// ---- POUs/Machine/UV_LED_Modul/FB_UvLedModule.TcPOU
FUNCTION_BLOCK FB_UvLedModule IMPLEMENTS I_DeviceBase
VAR_INPUT
  IbReady                  AT%I* : BOOL;
END_VAR

VAR_OUTPUT
  ObEnableHigh             AT%Q* : BOOL;
  ObLowIntenseMode         AT%Q* : BOOL;
  ObDisableLeft            AT%Q* : BOOL;
  ObDisableRight           AT%Q* : BOOL;
  OnIntensitySetpoint      AT%Q* : WORD;  (*Setpoint for intensity control  [digit]*)
END_VAR

VAR
  _bActivate                     : BOOL;
  _sName                         : STRING := '';
  _nColorRGB                     : UDINT;
  _sColorName                    : STRING := 'undef';    (*color name*)
END_VAR

VAR CONSTANT
  CnAnalogMinDigit               : DINT := 0;      (*Min value analog-output in digit*)
  CnAnalogMaxDigit               : DINT := 32767;  (*Max value analog-output in digit*)
  CnMinIntensitySetpoint         : DINT := 5;      (*Min setpoint for intensity control [%]*)
  CnMaxIntensitySetpoint         : DINT := 100;    (*Max setpoint for intensity control [%]*)
END_VAR

VAR PERSISTENT
  RbLowIntenseMode               : BOOL := FALSE;  (*Visu: set low intense mode*)
  RbDisableLeft                  : BOOL := FALSE;  (*Visu: disable left SLM*)
  RbDisableRight                 : BOOL := FALSE;  (*Visu: disable right SLM*)
  RnIntensitySetpoint            : DINT := 20;     (*Visu: setpoint for intensity control [%]*)
END_VAR

(*Set outputs*)
ObEnableHigh        := _bActivate;
ObLowIntenseMode    := RbLowIntenseMode;
ObDisableLeft       := RbDisableLeft;
ObDisableRight      := RbDisableRight;
OnIntensitySetpoint := DINT_TO_WORD(CnAnalogMaxDigit * RnIntensitySetpoint / 100);  (*Setpoint [digit]*)

METHOD Init : BOOL
VAR_INPUT
  nColorRGB    : UDINT;     (*color RGB*)
  sColorName   : STRING;    (*color name*)
END_VAR
_nColorRGB := nColorRGB;
_sColorName := sColorName;
END_METHOD

METHOD mDisable : BOOL
_bActivate := FALSE;
END_METHOD

METHOD mEnable : BOOL
_bActivate := TRUE;
END_METHOD

{attribute 'monitoring':='call'}
PROPERTY pActive : BOOL
GET
pActive := _bActivate;
END_GET
END_PROPERTY

PROPERTY pErrorCode : INT
GET
pErrorCode := 0;  // no error
END_GET
END_PROPERTY

END_FUNCTION_BLOCK

// ---- POUs/Print/Ads/FB_ADS_CAMERA.TcPOU
FUNCTION_BLOCK FB_ADS_CAMERA EXTENDS FB_AdsBlockBase
VAR
  stAds : ST_ADS_CAMERA;
END_VAR



// Todo redirect PucPath to internal sAdsStruct instead of fb Instance
// - write InstanceName
// - or override getPucPath() (but is PRIVATE)

// The output variables are not used, please add eaccessors if needed
(*
 (*Out*)
  iO_MaxNbMarksQV           : INT := GVL_Camera.cC_QUALIVISION_MAX_NB_MARKS; 
  sO_PointsReadQV           : ST_COMMAND_PLC;    (*New points read by QualiVision*)
  iO_AvailableNbReadPointQV : INT; 
  sO_ReadPointsQV           : ARRAY[1..GVL_Camera.cC_QUALIVISION_MAX_NB_MARKS] OF ST_CAMERA_CORRECTION_QV;
*)

{attribute 'monitoring' := 'call'}
(*
  Name of the block. 
  A friendly name (which is used in the PUC to show the element (only for some blocks/apps))
*)
PROPERTY aName : T_MaxString
GET
aName := aO_Name;
END_GET
SET
aO_Name := aName;
stAds.aO_Name := aName; // update in struct as well
END_SET
END_PROPERTY

PROPERTY bEnable : BOOL
GET
bEnable   := stAds.bI_Enable;   // Set ads interface variable
END_GET
SET
stAds.bI_Enable := bEnable;   // set interface variable
END_SET
END_PROPERTY

METHOD config
VAR_INPUT

END_VAR

//initRemVar();
END_METHOD

PROPERTY eCameraDevice : E_CameraDevice
GET
eCameraDevice := stAds.eI_CameraDevice;
END_GET
SET
stAds.eI_CameraDevice := eCameraDevice;
END_SET
END_PROPERTY

PROPERTY eCameraMode : E_CameraMode
GET
eCameraMode := stAds.eI_CameraMode;
END_GET
SET
stAds.eI_CameraMode := eCameraMode;
END_SET
END_PROPERTY

PROPERTY eTeachProgress : EN_CAMERA_TEACH
GET
eTeachProgress := stAds.eI_TeachProgress;
END_GET
END_PROPERTY

METHOD PROTECTED getPucPath : STRING
VAR
END_VAR
// apply puc path to struct (instead of fb declaraion)
getPucPath := F_Concat3(SUPER^.getPucPath(), '.', 'stAds');
END_METHOD

PROPERTY pCorrectionPointsIndication : POINTER TO ARRAY[1..4] OF ST_CORRECTION_POINT;
GET
pCorrectionPointsIndication := ADR(stAds.sI_CorrectionPointIndication);
END_GET
END_PROPERTY

PROPERTY pTeachPointsQV : POINTER TO ARRAY[1..GVL_Camera.cC_QUALIVISION_MAX_NB_MARKS] OF ST_CAMERA_TEACH_QV;
GET
pTeachPointsQV := ADR(stAds.sI_TeachPointsQV);
END_GET
END_PROPERTY

(*
  Setup constant ADS Block definitions.
  HOWTO: in abstract implmentation call
      init(aVersion:=, aType:=, nType:=, eLayer:=);
*)
METHOD  setup

init(aVersion:=convertVersionIntToString(stAds.iO_Version), aType:=stAds.aO_Type, nType:=ePr_BLK_CAMERA, eLayer:=E_AdsLayer.Structural);
END_METHOD

PROPERTY sMsgInterface : POINTER TO ST_ADS_MSG_IF
GET
sMsgInterface := ADR(stAds.sO_Message);
END_GET
END_PROPERTY

END_FUNCTION_BLOCK

// ---- POUs/Print/Ads/FB_ADS_DVTSHEETALIGNMENT.TcPOU
FUNCTION_BLOCK FB_ADS_DVTSHEETALIGNMENT EXTENDS FB_AdsBlockBase
VAR
  // ---------------------------------
  // ADS interface block specific
  sO_Message         : ST_ADS_MSG_IF;
  
  bI_Enable          : BOOL := TRUE;    (*Enable processing*)

  bI_UsePrintMark    : BOOL := TRUE;    (*Enable processing of print marks*)
  sI_PrintMarkSizeX  : ST_VAR_IN_REAL;  (*Print mark X size [mm]*)
  sI_PrintMarkSizeY  : ST_VAR_IN_REAL;  (*Print mark Y size [mm]*)

  sI_HeadGap         : ST_VAR_IN_REAL;  (*Gap between head and substrate [mm]*)

  lI_SegmentSize     : UDINT;           (*Distance between two images in pixel*)
  lI_SegmentCount    : UDINT;           (*Number of images*)
  fI_SegmentAngle    : REAL;            (*Angle between two segments in deg*)

  sI_DeltaX          : ST_VAR_IN_REAL;  (*X offset between camera marks [mm]*)

  bI_IsMaintenanceJob: BOOL;            (*Maintenance job: disable shift and rotation*)

  (*Out*)
  sO_CurrentAngle    : ST_VAR_OUT_REAL; (*Last measured angle in deg*)
  lO_CurrentYShift   : UDINT;           (*Last measured Y Shift in Pixel*)

  bO_RangeErrorAngle : BOOL;            (*Measured angle out of range*)
  bO_RangeErrorShift : BOOL;            (*Measured shift out of range*)

  // ---------------------------------
END_VAR
VAR PERSISTENT
  aR_Pattern         : UDINT;           (*check pattern for rem validity*)
  bR_Enable          : BOOL;            (*remanent: *)
  bR_UsePrintMark    : BOOL;            (*remanent: *)
  fR_PrintMarkSize_X : REAL;            (*remanent: *)
  fR_PrintMarkSize_Y : REAL;            (*remanent: *)
  fR_HeadGap         : REAL;            (*remanent: head gap in [mm]*)
  fR_DeltaX          : REAL;            (*remanent: *)
END_VAR

PROPERTY bEnable : BOOL
GET
bEnable   := bI_Enable;   // Set ads interface variable
bR_Enable := bI_Enable;   // Update remanent variable
END_GET
SET
bI_Enable := bEnable;   // set interface variable
bR_Enable := bEnable;   // update remanent variable
END_SET
END_PROPERTY

PROPERTY bIsMaintenanceJob : BOOL
GET
bIsMaintenanceJob := bI_IsMaintenanceJob;   // Set ads interface variable
END_GET
SET
bI_IsMaintenanceJob := bIsMaintenanceJob;   // Set ads interface variable
END_SET
END_PROPERTY

PROPERTY bRangeErrorAngle : BOOL
SET
bO_RangeErrorAngle := bRangeErrorAngle;
END_SET
END_PROPERTY

PROPERTY bRangeErrorShift : BOOL
SET
bO_RangeErrorShift := bRangeErrorShift;
END_SET
END_PROPERTY

PROPERTY bUsePrintMark : BOOL
GET
bUsePrintMark   := bI_UsePrintMark;   // Set ads interface variable
bR_UsePrintMark := bI_UsePrintMark;   // Update remanent variable
END_GET
SET
bI_UsePrintMark := bUsePrintMark;   // set interface variable
bR_UsePrintMark := bUsePrintMark;   // update remanent variable
END_SET
END_PROPERTY

METHOD config
VAR_INPUT
  bPrintMarkSizeX_Exist : BOOL;
  aPrintMarkSizeX_Unit  : STRING;
  fPrintMarkSizeX_Min   : REAL;
  fPrintMarkSizeX_Max   : REAL;
  
  bPrintMarkSizeY_Exist : BOOL;
  aPrintMarkSizeY_Unit  : STRING;
  fPrintMarkSizeY_Min   : REAL;
  fPrintMarkSizeY_Max   : REAL;
  
  bHeadGap_Exist        : BOOL;
  aHeadGap_Unit         : STRING;
  fHeadGap_Min          : REAL;
  fHeadGap_Max          : REAL;

  bDeltaX_Exist         : BOOL;
  aDeltaX_Unit          : STRING;
  fDeltaX_Min           : REAL;
  fDeltaX_Max           : REAL;
  
  bCurrentAngle_Exist   : BOOL;
  aCurrentAngle_Unit    : STRING;
  fCurrentAngle_Min     : REAL;
  fCurrentAngle_Max     : REAL;
END_VAR
sI_PrintMarkSizeX.bC_Exist := bPrintMarkSizeX_Exist;
sI_PrintMarkSizeX.aC_Unit  := aPrintMarkSizeX_Unit;
sI_PrintMarkSizeX.fC_Min   := fPrintMarkSizeX_Min;
sI_PrintMarkSizeX.fC_Max   := fPrintMarkSizeX_Max;
sI_PrintMarkSizeY.bC_Exist := bPrintMarkSizeY_Exist;
sI_PrintMarkSizeY.aC_Unit  := aPrintMarkSizeY_Unit;
sI_PrintMarkSizeY.fC_Min   := fPrintMarkSizeY_Min;
sI_PrintMarkSizeY.fC_Max   := fPrintMarkSizeY_Max;
sI_HeadGap.bC_Exist        := bHeadGap_Exist;
sI_HeadGap.aC_Unit         := aHeadGap_Unit;
sI_HeadGap.fC_Min          := fHeadGap_Min;
sI_HeadGap.fC_Max          := fHeadGap_Max;
sI_DeltaX.bC_Exist         := bDeltaX_Exist;
sI_DeltaX.aC_Unit          := aDeltaX_Unit;
sI_DeltaX.fC_Min           := fDeltaX_Min;
sI_DeltaX.fC_Max           := fDeltaX_Max;
sO_CurrentAngle.bC_Exist   := bCurrentAngle_Exist;
sO_CurrentAngle.aC_Unit    := aCurrentAngle_Unit;
sO_CurrentAngle.fC_Min     := fCurrentAngle_Min;
sO_CurrentAngle.fC_Max     := fCurrentAngle_Max;

sO_CurrentAngle.bC_Exist   := FALSE;

initRemVar();
END_METHOD

PROPERTY fDeltaX : REAL
GET
fDeltaX   := sI_DeltaX.fI_Val;   // Set ads interface variable
fR_DeltaX := sI_DeltaX.fI_Val;
END_GET
END_PROPERTY

// HeadGap in [mm]
PROPERTY fHeadGap : LREAL
GET
fHeadGap   := sI_HeadGap.fI_Val;   // Set ads interface variable
fR_HeadGap := sI_HeadGap.fI_Val;   // Update remanent variable
END_GET
SET
sI_HeadGap.fI_Val := TO_REAL(fHeadGap);   // set interface variable
fR_HeadGap        := TO_REAL(fHeadGap);   // update remanent variable
END_SET
END_PROPERTY

PROPERTY fMarkSizeX : REAL
GET
fMarkSizeX         := sI_PrintMarkSizeX.fI_Val;   // Set ads interface variable
fR_PrintMarkSize_X := sI_PrintMarkSizeX.fI_Val;   // Update remanent variable
END_GET
END_PROPERTY

PROPERTY fMarkSizeY : REAL
GET
fMarkSizeY         := sI_PrintMarkSizeY.fI_Val;   // Set ads interface variable
fR_PrintMarkSize_Y := sI_PrintMarkSizeY.fI_Val;   // Update remanent variable
END_GET
END_PROPERTY

PROPERTY fO_CurrentAngle : LREAL
SET
sO_CurrentAngle.fO_Val := tO_REAL(fO_CurrentAngle);
END_SET
END_PROPERTY

PROPERTY fSegmentAngle : REAL
GET
fSegmentAngle := fI_SegmentAngle;   // Set ads interface variable
END_GET
END_PROPERTY

METHOD PROTECTED initRemVar
(*load default initial values if pattern was invalid*)
IF aR_Pattern <> 16#ABCD THEN
  aR_Pattern  := 16#ABCD;  
  bR_Enable   := TRUE;
  bR_UsePrintMark := 0;
  fR_PrintMarkSize_X := 0;
  fR_PrintMarkSize_Y := 0;
  fR_HeadGap  := 2;
  fR_DeltaX := 0;
END_IF

bI_Enable := bR_Enable;
bI_UsePrintMark := bR_UsePrintMark;
sI_PrintMarkSizeX.fI_Val := fR_PrintMarkSize_X;
sI_PrintMarkSizeY.fI_Val := fR_PrintMarkSize_Y;
sI_HeadGap.fI_Val := fR_HeadGap;
sI_DeltaX.fI_Val := fR_DeltaX;
END_METHOD

PROPERTY nO_CurrentYShift : UDINT
SET
lO_CurrentYShift := nO_CurrentYShift;
END_SET
END_PROPERTY

PROPERTY nSegmentCount : UDINT
GET
nSegmentCount := lI_SegmentCount;   // Set ads interface variable
END_GET
END_PROPERTY

PROPERTY nSegmentSize : UDINT
GET
nSegmentSize := lI_SegmentSize;   // Set ads interface variable
END_GET
END_PROPERTY

(*
  Setup constant ADS Block definitions.
  HOWTO: in abstract implmentation call
      init(aVersion:=, aType:=, nType:=, eLayer:=);
*)
METHOD  setup
init(aVersion:='01.00.10', aType:='DvtSheetAlignment', nType:=ePr_BLK_SA, eLayer:=E_AdsLayer.Structural);
END_METHOD

PROPERTY sMsgInterface : POINTER TO ST_ADS_MSG_IF
GET
sMsgInterface := ADR(sO_Message);
END_GET
END_PROPERTY

END_FUNCTION_BLOCK

// ---- POUs/Print/Camera/FB_CameraBase.TcPOU
(*
  Base camera system
  Implements I_Camera: set I_CameraSink.   
*)
FUNCTION_BLOCK ABSTRACT FB_CameraBase EXTENDS FB_Commons IMPLEMENTS I_Camera, I_CameraTriggerDevice

VAR
  _bInitialized             : BOOL;
  _iCameraSink              : I_CameraSink;
  _iCameraTrigger           : I_CameraTrigger;
  _bSimulate                : BOOL;
  _nPrintUnitResolution     : UDINT;           (*printhead pixel resolution [dpi]*)
  _nPrintUnitSubPx          : UDINT;           (*print unit SubPixel resolution [SubPx]*)
  _bUseCameraTrigger        : BOOL;            (*use a trigger output timestamp I/O*)
  _bUseCameraTriggerFeedback : BOOL;           (*use a camera triggered feedback timestamp I/O*)
  _eCameraMode              : E_CameraMode;    (*desired camera mode*)
  _ePossibleMode            : E_CameraMode;    (*currently possible mode*)
  _fSubstrateLength         : LREAL := 1;      (*Substrate length [m]*)
  _fSubstrateWidth          : LREAL := 1;      (*Substrate width [m]*)
  _fImageLength             : LREAL := 1;      (*Image length [m]*)
  _fImageWidth              : LREAL := 1;      (*Image width [m]*)
  _fFrameLength             : LREAL := 1;      (*Camera Frame width in [px]*)
  _bActivated               : BOOL;            (*Camera is activated*)
  _sVisuName                : STRING := 'unvailable';     (*detail visualisation instance name*)
  
  // status
  _bCamTriggerOk            : BOOL;
  _bCamTriggerStarted       : BOOL;
  _bCamTriggerDone          : BOOL;   
  _nCamStartPos             : DINT;            (*Cam start position ideal [SubPx]*)
  _nCamStartPosDeviation    : DINT;            (*Cam stated position real [SubPx]*)
  _nRxCamPoints             : UDINT;           (*number of received cam points*)

  // helper
  stCamPoint                : ST_DeformationPointAccurate;(*actual camera point*)
    
  // messaging
  _pMsgConfig               : POINTER TO CalmarCommons.ST_MSG_CONFIG;
END_VAR

VAR PERSISTENT
  _fTriggerDistance         : LREAL;           (*[m] Distance between Sensor and Trigger*)
  _fTriggerPulseLength      : LREAL := 10;     (*[ms] Length of trigger signal in ms, min. 3 bus cycles*)
  _fDetectToCameraOffset    : LREAL := 0.1;    (*[m] Distance between input trigger and camera, mech.*)
  _fCameraToPrintOffset     : LREAL := 0.0;    (*[m] Distance between Camera and PU, mech, This offset can be used to shift the reference of a camera/sheet-detect, e.g. because this reference is different from to one where the alignment Camera/sheetdetect-PrintUnit has been made*)
END_VAR

METHOD ActivateCam : BOOL
VAR_INPUT
  iCameraSink : I_CameraSink;
END_VAR
IF iCameraSink = 0 THEN
  LogError('Invalid parameter (0 pointer)');
  ActivateCam := FALSE;
  RETURN; 
ELSIF _iCameraSink <> 0 AND iCameraSink <>_iCameraSink THEN
  LogError('SetSink failed: other sink already exists');
  ActivateCam := FALSE;
  RETURN; 
END_IF 

_iCameraSink := iCameraSink;
_iCameraTrigger.Enable(iCam:=THIS^, bUseCameraTrigger:=_bUseCameraTrigger, bUseCameraTriggerFeedback:=_bUseCameraTriggerFeedback);

_bActivated := TRUE;
ActivateCam:=TRUE;
END_METHOD

(*
  Activate/Deactivate camera trigger device
*)
PROPERTY bEnableTrigger : BOOL
SET
IF bEnableTrigger THEN
  _iCameraTrigger.Enable(iCam := THIS^, bUseCameraTrigger:= _bUseCameraTrigger, bUseCameraTriggerFeedback:=_bUseCameraTriggerFeedback);
ELSE
  _iCameraTrigger.Disable();
END_IF
END_SET
END_PROPERTY

(*
  Activate/Deactivate camera manual teach mode
*)
PROPERTY bManualTeach : BOOL
SET
_iCameraTrigger.bManualTeach := bManualTeach;
END_SET
END_PROPERTY

{attribute 'monitoring':='call'}
PROPERTY bSimulate : BOOL
GET
bSimulate := _bSimulate;
END_GET
SET
_bSimulate := bSimulate;
END_SET
END_PROPERTY

METHOD CamTrigger
VAR_INPUT
  bOk             : BOOL;     // trigger is ok
	nPos            : DINT;     // camera triggered position
  nPosDeviation   : DINT;     // camera started deviation
  nX0             : DINT;     // detected position sheet/repetition
END_VAR
_nRxCamPoints := 0;
_bCamTriggerStarted    := TRUE;
_bCamTriggerDone       := FALSE;
_bCamTriggerOk  := bOk;
_nCamStartPos   := nPos;
_nCamStartPosDeviation := nPosDeviation;

LogLvl(Lvl:=E_LogSeverity.Debug, Msg:=F_Concat2('CamTrigger at X0=', TO_STRING(nPos)));
IF _iCameraSink <> 0 THEN   // inform sink
  _iCameraSink.CamStarted(nX0:=nX0);
END_IF
END_METHOD

METHOD CamTriggerDone
_bCamTriggerStarted    := FALSE;  // this call marks the end of the camera trigger period
_bCamTriggerDone       := TRUE;

LogLvl(Lvl:=E_LogSeverity.Debug, Msg:='CamTriggerDone');
IF _iCameraSink <> 0 THEN   // inform sink
  _iCameraSink.CamDone();
END_IF
END_METHOD

METHOD DeactivateCam : BOOL
VAR_INPUT
  iSink : I_CameraSink;
END_VAR
IF _iCameraSink <> 0 AND iSink <> _iCameraSink THEN
  LogError('remove sink failed: inconsistent');
  DeactivateCam := FALSE;
  RETURN;  
END_IF

_iCameraSink := 0;
_iCameraTrigger.Disable();
_bActivated := FALSE;
DeactivateCam:=TRUE;
END_METHOD

{attribute 'monitoring':='call'}
PROPERTY ABSTRACT eCameraMode : E_CameraMode
GET
END_GET
END_PROPERTY

{attribute 'monitoring':='call'}
PROPERTY ABSTRACT eDeviceType : E_CameraDevice
GET
END_GET
END_PROPERTY

{attribute 'monitoring':='call'}
PROPERTY fCameraToPrintOffset : LREAL
GET
//This offset can be used to shift the reference of a camera, e.g. because this reference is different from to one where the alignment Camera-PrintUnit has been made
fCameraToPrintOffset := _fCameraToPrintOffset;
END_GET
SET
_fCameraToPrintOffset := fCameraToPrintOffset;
END_SET
END_PROPERTY

{attribute 'monitoring':='call'}
PROPERTY fDetectToCameraOffset : LREAL
GET
//This offset can be used to shift the reference of a camera, e.g. because this reference is different from to one where the alignment Camera-PrintUnit has been made
fDetectToCameraOffset := _fDetectToCameraOffset;
END_GET
SET
_fDetectToCameraOffset := fDetectToCameraOffset;
END_SET
END_PROPERTY

{attribute 'monitoring':='call'}
(* camera frame size in [px]*)
PROPERTY fFrameLength : LREAL
GET
fFrameLength := _fFrameLength;
END_GET
SET
_fFrameLength := fFrameLength;
END_SET
END_PROPERTY

{attribute 'monitoring':='call'}
(*Image Length/Depth in [m]*)
PROPERTY fImageLength : LREAL
GET
fImageLength := _fImageLength;
END_GET
SET
_fImageLength := fImageLength;
END_SET
END_PROPERTY

{attribute 'monitoring':='call'}
(*Image Width in [m]*)
PROPERTY fImageWidth : LREAL
GET
fImageWidth := _fImageWidth;
END_GET
SET
_fImageWidth := fImageWidth;
END_SET
END_PROPERTY

{attribute 'monitoring':='call'}
(*Substrate Length/Depth in [m]*)
PROPERTY fSubstrateLength : LREAL
GET
fSubstrateLength := _fSubstrateLength;
END_GET
SET
//ROI in Print direction
IF _iCameraTrigger <> 0 THEN
  _iCameraTrigger.SetSubstrateLength(fSubstrateLength := fSubstrateLength);   // save to camera trigger
  _fSubstrateLength := fSubstrateLength;                                      // save to camera
END_IF
END_SET
END_PROPERTY

{attribute 'monitoring':='call'}
(*Substrate Width in [m]*)
PROPERTY fSubstrateWidth : LREAL
GET
fSubstrateWidth := _fSubstrateWidth;
END_GET
SET
_fSubstrateWidth := fSubstrateWidth;
END_SET
END_PROPERTY

{attribute 'monitoring':='call'}
PROPERTY fTriggerDistance : LREAL
GET
fTriggerDistance := _fTriggerDistance;
END_GET
SET
_fTriggerDistance := fTriggerDistance;
END_SET
END_PROPERTY

PROPERTY fTriggerPulseLength : LREAL
GET
fTriggerPulseLength := _fTriggerPulseLength;
END_GET
END_PROPERTY

METHOD ABSTRACT GetCamStatus : BOOL
VAR_OUTPUT
  bConnectionOK  : BOOL;    // Camera connected
  bTeachOk       : BOOL;    // Teach successful
  nTeachedPoints : UDINT;   // Teached points for this job
  nScannedPoints : UDINT;   // Scanned points on current sheet  
  bCamStarted    : BOOL;    // Camera trigger is active, cam started
  bCamDone       : BOOL;    // Camera finished on last CT
  bErrors        : ARRAY[1..GVL_Camera.nC_NbCamErrors] OF BOOL;  // generic error flag list
END_VAR
END_METHOD

METHOD Init
VAR_INPUT
  nPrintUnitResolution         : UDINT;    (*printhead pixel resolution [dpi]*)
  nPrintUnitSubPx              : UDINT;    (*print unit subPixel resolution [SubPx]*)
  iCameraTrigger               : I_CameraTrigger;
  bUseCameraTrigger            : BOOL;     (*use a trigger output timestamp I/O*)
  bUseCameraTriggerFeedback    : BOOL;     (*use a camera triggered feedback timestamp I/O*)
END_VAR
IF nPrintUnitResolution <> 0 AND iCameraTrigger <> 0 THEN
  _nPrintUnitResolution := nPrintUnitResolution;
  _nPrintUnitSubPx      := nPrintUnitSubPx;
  _iCameraTrigger       := iCameraTrigger;
  
  _bUseCameraTrigger := bUseCameraTrigger;
  _bUseCameraTriggerFeedback := bUseCameraTriggerFeedback;
  
  _bInitialized := TRUE;
ELSE
  _bInitialized := FALSE;
END_IF
END_METHOD

METHOD mJobStart : BOOL
END_METHOD

(*
  Set mode to camera.
  :return: TRUE if success
*)
METHOD ABSTRACT setCameraMode : BOOL
VAR_INPUT
  eCameraMode : E_CameraMode;
END_VAR
END_METHOD

METHOD setMsgInterface : BOOL
VAR_INPUT
	pMsgConfig	: POINTER TO CalmarCommons.ST_MSG_CONFIG;
END_VAR
_pMsgConfig := pMsgConfig;
END_METHOD

{attribute 'monitoring':='call'}
PROPERTY sName : STRING
GET
sName := 'undefined';
END_GET
END_PROPERTY

{attribute 'monitoring':='call'}
PROPERTY sVisuName : STRING
GET
sVisuName := _sVisuName;
END_GET
SET
_sVisuName := sVisuName;
END_SET
END_PROPERTY

END_FUNCTION_BLOCK

// ---- POUs/Print/Camera/FB_CameraDummy.TcPOU
FUNCTION_BLOCK FB_CameraDummy EXTENDS FB_CameraBase
VAR_INPUT
END_VAR
VAR_OUTPUT
END_VAR
VAR
END_VAR

{attribute 'monitoring':='call'}
PROPERTY eCameraMode : E_CameraMode
GET
eCameraMode := _eCameraMode;
IF _eCameraMode = E_CameraMode.Auto THEN
  eCameraMode := E_CameraMode.NoCorrection;
END_IF
END_GET
END_PROPERTY

PROPERTY eDeviceType : E_CameraDevice
GET
eDeviceType := E_CameraDevice.SheetDetect;
END_GET
END_PROPERTY

METHOD GetCamStatus : BOOL
VAR_OUTPUT
  bConnectionOK  : BOOL;    // Camera connected
  bTeachOk       : BOOL;    // Teach successful
  nTeachedPoints : UDINT;   // Teached points for this job
  nScannedPoints : UDINT;   // Scanned points on current sheet
  bCamStarted    : BOOL;    // Camera trigger is active, cam started
  bCamDone       : BOOL;    // Camera finished on last CT
  bErrors        : ARRAY[1..GVL_Camera.nC_NbCamErrors] OF BOOL;  // generic error flag list
END_VAR
bConnectionOK  := TRUE;  //NO comm with a cam 
bTeachOk       := TRUE;  //NO teach availabe
nTeachedPoints := 0;
nScannedPoints := 0;
bCamStarted    := _bCamTriggerStarted;
bCamDone       := _bCamTriggerDone;

GetCamStatus := TRUE;
END_METHOD

(*
  Set mode to camera.
  :return: TRUE if success
*)
METHOD setCameraMode : BOOL
VAR_INPUT
  eCameraMode : E_CameraMode;
END_VAR
IF eCameraMode = E_CameraMode.NoCorrection THEN   // supported mode
  
  _eCameraMode := eCameraMode; 
  setCameraMode := TRUE;        // set desired mode
ELSE
  LogError(F_Concat3('Camera mode=', TO_STRING(eCameraMode), ' not supported by camera'));
  _eCameraMode := E_CameraMode.NoCorrection;
END_IF
END_METHOD

{attribute 'monitoring':='variable'}
PROPERTY sName : STRING
GET
sName := 'SheetDetect';
END_GET
END_PROPERTY

END_FUNCTION_BLOCK

// ---- POUs/Print/Camera/FB_CameraTcpIp.TcPOU
(*
  Base camera system with TcpIp communicatiom
  Implements callback function (rx_callback) for received TcpIp messages.   
*)
FUNCTION_BLOCK ABSTRACT FB_CameraTcpIp EXTENDS FB_CameraBase IMPLEMENTS I_TcpIp_RxMsgHandler

VAR
  sLastMessage              : STRING(GVL_TcpIp.TCP_RXDATA_SIZE);          (*rx telegram string*)
  nLastMessageSz            : UDINT;                                      (*receive message length *)
  sMemLastMessage           : STRING(GVL_TcpIp.TCP_RXDATA_SIZE);          (*mem rx telegram string*)
  nRxMsg                    : UDINT;                (*rx telegram counter*)
  bMsgReceived              : BOOL;                 (*we received a message*)
  sState                    : STRING;               (*state change event as string*)

  sLastErrorMessage         : STRING(GVL_TcpIp.TCP_RXDATA_SIZE);          (*rx telegram error string*)
  _bConnectionError         : BOOL;
  _pFbTcpIpClient           : POINTER TO FB_TcpClient;
END_VAR

METHOD ActivateCam : BOOL
VAR_INPUT
  iCameraSink : I_CameraSink;
END_VAR
ActivateCam := SUPER^.ActivateCam(iCameraSink:=iCameraSink);

IF _pFbTcpIpClient = 0 THEN
  LogError('No tcpip client assigned');
  ActivateCam := 0;
  RETURN;
END_IF

_pFbTcpIpClient^.bEnable := TRUE;
END_METHOD

PROPERTY bConnectionErr : BOOL
GET
IF _pFbTcpIpClient = 0 THEN RETURN; END_IF

_bConnectionError := FALSE;
IF _bActivated THEN
  IF NOT _pFbTcpIpClient^.bConnected OR _pFbTcpIpClient^.bError THEN
    bConnectionErr := TRUE;
    _bConnectionError := TRUE;
  END_IF 
END_IF
END_GET
END_PROPERTY

METHOD DeactivateCam : BOOL
VAR_INPUT
  iSink : I_CameraSink;
END_VAR
DeactivateCam := SUPER^.DeactivateCam(iSink:=iSink);

IF _pFbTcpIpClient = 0 THEN
  LogError('No tcpip client assigned');
  DeactivateCam := 0;
  RETURN;
END_IF

_pFbTcpIpClient^.bEnable := FALSE;
END_METHOD

METHOD ABSTRACT GetCamStatus : BOOL
VAR_OUTPUT
  bConnectionOK  : BOOL;    // Camera connected
  bTeachOk       : BOOL;    // Teach successful
  nTeachedPoints : UDINT;   // Teached points for this job
  nScannedPoints : UDINT;   // Scanned points on current sheet
  bCamStarted    : BOOL;    // Camera trigger is active, cam started
  bCamDone       : BOOL;    // Camera finished on last CT
  bErrors        : ARRAY[1..GVL_Camera.nC_NbCamErrors] OF BOOL;  // generic error flag list
END_VAR
END_METHOD

METHOD rx_callback
VAR_INPUT
	sMessage	: CalmarCompTcpIp.ST_TcpMsg;
END_VAR
sLastMessage  := sMessage.sMessage;   // store message locally
nRxMsg        := nRxMsg + 1;
nLastMessageSz := LEN2(ADR(sLastMessage));

bMsgReceived  := TRUE;
END_METHOD

METHOD setTcpIpClient : BOOL
VAR_INPUT
  pTcpIpClient  : POINTER TO FB_TcpClient;
END_VAR
_pFbTcpIpClient := pTcpIpClient;
END_METHOD

METHOD state_callback
VAR_INPUT
	(* state change event as string (think to convert it to an enum for easier handling later)*)
	state	: STRING;
END_VAR
sState := state;   // store state locally
END_METHOD

END_FUNCTION_BLOCK

// ---- POUs/Print/Camera/FB_CameraTrigger.TcPOU
FUNCTION_BLOCK FB_CameraTrigger EXTENDS FB_Commons IMPLEMENTS I_CameraTrigger, I_StartPosDetect
(*************************************************************************************************)
(*  FILENAME:    FB_CameraTrigger                                                                *)
(*  PROJECT:     CALMAR PUPLC                                                                    *)
(*  COPYRIGHT:   All rights reserved (c) Wifag//Polytype, Fribourg/Switzerland (2016)            *)
(*  ENVIRONMENT: TwinCAT PLC                                                                     *)
(*  VERSION:     <version>                                                                       *)
(*************************************************************************************************)
(*  DESCRIPTION:                                                                   <description> *)
(*    Generate timestamp trigger output based on timestamp sensor input. Two variants            *)
(*    exist, a timebased approach where the trigger time is calculated at the time the sensor    *)
(*    event occurs, and a second approach where the sensor event time is translated to a sensor  *)
(*    event position, and a trigger is generated when the calculated trigger position has almost *)
(*    been reached. The second approach has the advantage that is is less susceptible to speed   *)
(*    variations.                                                                                *)
(*                                                                                </description> *)
(*************************************************************************************************)

{library public}
VAR_INPUT
  bI_HwEnable                             : BOOL;            // relase (enable SheetDetect) from machine
  bI_AutomaticMode                        : BOOL;            // machine is in automatic mode
  (* - (EL1252) StartPosition detect sensor*)
  bI_SensorSupervisionEnable              : BOOL := TRUE;    // enable SheetDetect with supervision 
  bI_Sensor_State                   AT%I* : BOOL;            // Sensor signal
  tI_Sensor_TimeStampPos            AT%I* : T_DCTIME64;      // Sensor last detection timestamp
  (* - (EL1252) Camera started feedback trigger/signal*)
  bI_TriggerFeedback_State          AT%I* : BOOL;           // Sensor signal
  tI_TriggerFeedback_TimeStampPos   AT%I* : T_DCTIME64;     // Sensor last detection timestamp

  (*System signals*)
  iI_CurrentPos                   : DINT;                   // Current position in [SubPx]*)
  fI_ConveyorSpeed                : LREAL;                  // Current speed of substrate in [m/s]*)
  
  (*Debug & Test*)
  bI_ManualTrigger                : BOOL;                   // Manual start trigger
END_VAR

VAR_OUTPUT
  (*Link to EL2252*)
  ObTrigger                 AT%Q* : BOOL;                   // EL2252 Output1 - TRUE=start camer
  OtTriggerStartTime        AT%Q* : T_DCTIME64;             // EL2252 Timestamp - where to set outputs
  OnTriggerCommand          AT%Q* : BYTE;                   // EL2252 Command - activation timestamp ouput
END_VAR

(*{library private}*)
VAR
  bInitOk                         : BOOL;           // initialized
  bSpeedValid                     : BOOL;           // speed is valid
  bTriggerEnabled                 : BOOL;           // detection & trigger is enabled
  bTriggerArmed                   : BOOL;           // trigger is armed
  bCamValid                       : BOOL;           // camera is valid
  bTriggerOk                      : BOOL;
  rT_Sensor                       : R_TRIG;        // rising edge trigger sensor
  
  (*configuration*)
  _nResolution                    : INT := 1;       // Printhead Resolution [e.g. 600] x Subpixel Resolution [e.g. 32]*)
  _bUsePositionTrigger            : BOOL;           // FALSE: Calculate time with speed and position distance@sensor event, TRUE: Calculate sensor event position, launch trigger based on position
  _bUseCameraTrigger              : BOOL;           // (cam specific setting) Generate camera trigger output
  _bUseCameraTriggerFeedback      : BOOL;           // (cam specific setting) Evaluate camera triggered feedback
  _bCamManualTeachMode            : BOOL;           // cam in manual teach mode
  _tMemTriggerFeedback_TimeStampPos : T_DCTIME64;
  _nSubstrateLength               : DINT;           // Substrate length in pulse [SubPx]
  _fSubstrateLength               : LREAL;          // Substrate length in [m]
  _fTriggerDistance               : LREAL;          // Distance between Sensor and Trigger [m]
  _fTriggerLength                 : LREAL := 10;    // Length of trigger signal in ms, min. 3 bus cycles
  
  iActiveCam	                    : I_CameraTriggerDevice;  // active camera interface
  
  bSheetDetected                  : BOOL;
  bInhibitTrigger                 : BOOL;            (*inhibit trigger signals, TRUE=inhibit*)
  bReleaseInhibitTrigger          : BOOL;            (*condition to release inhibit trigger*)

  eState                          : BYTE;            (*State*)
  tSensor_TimeStamp               : T_DCTIME64;      (*Sensor last detection timestamp*)
  tTriggerFeedback_TimeStamp      : T_DCTIME64;      (*Trigger feedback last detection timestamp*)
  tCurrentTime                    : T_DCTIME64;      (*Current system dc time [64bit]*)
  tTrigger_EventTime              : T_DCTIME64;      (*Trigger event timestamp*)

  _bManualStart                   : BOOL;
  fDeltaDistance                  : LREAL;           (*Distance that the substrate moved between the detection and the treatment of the information [m]*)
  _nX0                            : DINT;            (*Detected X0 position of CT [SubPx] by sensor*)
  _nCamStartPos                   : DINT;            (*Camera start position*)
  _nCamStartedPos                 : DINT;            (*Camera started position [SubPx]*)
  
  tCurrentTimeStamp               : T_DCTIME64;      (* Get Current Timestamp *)
  tLastTimeStamp                  : T_DCTIME64;      (* Get Current Timestamp *)
  fCycleTime                      : LREAL;           (* Current calculated cycle time [s]*)

  fRemDist                        : LREAL;           (*Remaining distance until trigger occurs [m]*)
  fPreTriggerPosition             : LREAL;           (*Margin between effective trigger position and generation of timestamp*)

  (*Debug*)
  _bVerbose                       : BOOL;
END_VAR

VAR CONSTANT
  fC_MIN_CONVEYOR_SPEED           : LREAL := 0.01;
  fC_PreTrigFactor                : LREAL := 3.0;
  fC_SheetLengthMargin            : LREAL := 0.01;   (*Added 10 mm margin for substrate length in case of print quality strips at the end of sheet in case of start with edge*)
  fC_MaxCameraFeedbackTimeout     : LREAL := 28.0;   (*[ns] Max. timeout waiting for camera trigger feedback signal*)

  (*State*)
  cL_IDLE                         : BYTE := 0;       (*Idle state, no trigger active*)
  cL_SENSOREVENT                  : BYTE := 1;       (*Sensor started trigger generation*)
  cL_WAITALMOSTSTART              : BYTE := 2;       (*Wait timestamp calculation critera*)
  cL_WAITSTART                    : BYTE := 3;       (*Wait for trigger generation critera*)
  cL_WAITFEEDBACK                 : BYTE := 4;       (*Wait on feedback from trigger*)
  cL_TRIGACTIVE                   : BYTE := 5;       (*Trigger set*)
  cL_WAITSTOP                     : BYTE := 6;       (*Trigger reset*)

  (*EL2252 Command*)
  nC_EL2252Cmd_INACTIVE           : BYTE := 0;
  nC_EL2252Cmd_ACTIVE             : BYTE := 3;
END_VAR

IF NOT bInitOk THEN RETURN; END_IF;

// General calculations
bSpeedValid   := fI_ConveyorSpeed > fC_MIN_CONVEYOR_SPEED;    // speed valid (ignore trigger if not moving)
bCamValid     := SEL(iActiveCam<>0, FALSE, TRUE);             // camera valid (ignore trigger otherwise)
tCurrentTime  := F_GetCurDcTaskTime64();                      // current dc time (most accurate time stamp we have)
fCycleTime    := (TO_LREAL(tCurrentTime) - TO_LREAL(tLastTimeStamp)) * 1E-9;  tLastTimeStamp  := tCurrentTime;  // calculate cycle time of this block
bSheetDetected:= FALSE;                                       // Set to true below just for one cycle
bTriggerEnabled := bSpeedValid AND bI_HwEnable AND (bI_AutomaticMode OR _bCamManualTeachMode);
bTriggerArmed :=  NOT bInhibitTrigger AND bTriggerEnabled;
rT_Sensor(CLK := bI_Sensor_State AND bI_SensorSupervisionEnable);

// apply parameter
IF bCamValid THEN    // save dynamic changable settings
  _fTriggerDistance := iActiveCam.fTriggerDistance;
  _fTriggerLength   := iActiveCam.fTriggerPulseLength;
END_IF

// - Release inhibit trigger
bReleaseInhibitTrigger := bInhibitTrigger AND (iI_CurrentPos - (_nX0 + _nSubstrateLength)) > 0;
IF bReleaseInhibitTrigger THEN bInhibitTrigger := FALSE; END_IF

// Reset trigger if deactivated - should improve hanging triggers
IF NOT bTriggerEnabled AND eState > cL_IDLE THEN
  Reset();
  RETURN;
END_IF


(*State Machine ----------------------------------------------------------------*)
CASE eState OF
  cL_IDLE:     (*Not started, waiting for start trigger*)
  
    IF bTriggerArmed THEN (*ignore trigger else*)
 
      IF rT_Sensor.Q AND (bCamValid OR _bCamManualTeachMode) THEN      (*Start launched*)
        eState            := cL_SENSOREVENT;
        tSensor_TimeStamp := tI_Sensor_TimeStampPos;
        _bManualStart := FALSE;
        IF _bCamManualTeachMode THEN LogWarning('StartTrigger in manual teach mode'); END_IF
      ELSIF (bI_ManualTrigger AND bCamValid) THEN  (*Manual start launched*)
        eState            := cL_SENSOREVENT;
        tSensor_TimeStamp := tCurrentTime;
        _bManualStart := TRUE;
      ELSIF (rT_Sensor.Q OR bI_ManualTrigger) AND NOT bCamValid THEN   (*Trigger without active camera*)
        LogWarning('No camera or start device active, ignore trigger');
      END_IF;
      
    END_IF
    
    OnTriggerCommand := nC_EL2252Cmd_INACTIVE;
    ObTrigger        := FALSE;

  cL_SENSOREVENT:     (*Not started*)
    IF NOT bSpeedValid THEN 
      Reset();        // ignore trigger if not moving anymore (avoid zero division)
    ELSE
      (*Distance in [m] that the substrate has traveled between the sensor detection (time) current plc cycle*)
      fDeltaDistance     := UINT64_TO_LREAL(UInt64Sub64(ULINT_TO_ULARGE(tCurrentTime), ULINT_TO_ULARGE(tSensor_TimeStamp))) * 1E-9 * fI_ConveyorSpeed;
      (*Position where the sheet has been detected in [SubPx]*)
      _nX0               := iI_CurrentPos - F_MeterToSubPixel(fPosMeter:=fDeltaDistance, fResoSubPx:=_nResolution);
      
      IF _bUsePositionTrigger OR NOT _bUseCameraTrigger THEN
        eState             := cL_WAITALMOSTSTART;
      ELSE
        eState             := cL_WAITSTART;
        tTrigger_EventTime := (tSensor_TimeStamp + LREAL_TO_ULINT(_fTriggerDistance / fI_ConveyorSpeed * 1E9));
      END_IF;
      
      OnTriggerCommand := nC_EL2252Cmd_INACTIVE;
      ObTrigger         := TRUE;
      bInhibitTrigger   := TRUE;
      bSheetDetected    := TRUE;
      
    END_IF

  cL_WAITALMOSTSTART: (*Only active when bI_UsePositionTrigger=TRUE: wait until Start position almost reached, then set timestamp*)
    (*Remaining distance in [m], converted to REAL to avoid integer wrap problems*)
    fRemDist             := _fTriggerDistance + (DINT_TO_REAL(_nX0) - DINT_TO_REAL(iI_CurrentPos))*0.0254 / INT_TO_REAL(_nResolution);
    fPreTriggerPosition  := fC_PreTrigFactor * fCycleTime * fI_ConveyorSpeed;

    IF fRemDist < fPreTriggerPosition THEN
      eState             := cL_WAITSTART;
      tTrigger_EventTime := (tSensor_TimeStamp + LREAL_TO_ULINT(fRemDist / fI_ConveyorSpeed * 1E9));    // division save because we are moving to reach this position
      IF _bUseCameraTrigger AND NOT _bManualStart THEN
        OnTriggerCommand := nC_EL2252Cmd_ACTIVE;  (*Arm EL2252*)
      END_IF
      LogTsDiff(aIdent:= 'WAITALMOSTSTART: ', t1:=tTrigger_EventTime, t2:=tCurrentTime);
    ELSE
      eState           := cL_WAITALMOSTSTART;
      OnTriggerCommand := nC_EL2252Cmd_INACTIVE;
    END_IF;
    ObTrigger          := TRUE;

  cL_WAITSTART:       (*Wait until start time reached*)
    bTriggerOk := TRUE;
    IF (tTrigger_EventTime < tCurrentTime) THEN (* StartTime elapsed *)
      // position reached
      IF _bUseCameraTriggerFeedback THEN
        eState         := cL_WAITFEEDBACK;
      ELSE
        eState         := cL_TRIGACTIVE;
        iActiveCam.CamTrigger(bOk:=bTriggerOk, nPos:=iI_CurrentPos, nPosDeviation:=0, nX0:=_nX0);
      END_IF

      OnTriggerCommand := nC_EL2252Cmd_INACTIVE; (*Disarm already command to EL2252, trigger generated*)
    ELSE
      // position not yet reached
      eState           := cL_WAITSTART;
      IF _bUseCameraTrigger AND NOT _bManualStart THEN
        OnTriggerCommand := nC_EL2252Cmd_ACTIVE;  (*Arm EL2252*)
      END_IF
    END_IF;

    ObTrigger      := TRUE;  
    
  cL_WAITFEEDBACK:
    IF _bManualStart THEN //Simulate feedback in case of manual start
      tTriggerFeedback_TimeStamp:= tTrigger_EventTime + LREAL_TO_ULINT(1000.0 * 1E3); //Trigger event plus 1000ns
    ELSE
      IF tI_TriggerFeedback_TimeStampPos = _tMemTriggerFeedback_TimeStampPos AND tCurrentTime > (tTrigger_EventTime + LREAL_TO_ULINT(fC_MaxCameraFeedbackTimeout * 1E3)) THEN
        // feedback was not received in next plc cycle (timeout jitter in camera max. 28us)
        LogError(F_Concat3('No Camera trigger feedback received (timeout), after ', TO_STRING(TO_LREAL(tCurrentTime-tTrigger_EventTime)/1E6), 'ms'));
        bTriggerOk := FALSE;
        tTriggerFeedback_TimeStamp:= tTrigger_EventTime + LREAL_TO_ULINT(fC_MaxCameraFeedbackTimeout * 1E3);
      ELSE
        tTriggerFeedback_TimeStamp:= tI_TriggerFeedback_TimeStampPos;
			END_IF
    END_IF
    
  (*feedback signal is a very short trigger that the PLC sometimes cannot register, therefore we use the timestamp*)
    IF (tTriggerFeedback_TimeStamp <> _tMemTriggerFeedback_TimeStampPos) AND (tTriggerFeedback_TimeStamp > 0) OR _bManualStart THEN
      eState          := cL_TRIGACTIVE;
      // start position requested
      fDeltaDistance  := UINT64_TO_LREAL(UInt64Sub64(ULINT_TO_ULARGE(tCurrentTime), ULINT_TO_ULARGE(tTrigger_EventTime))) * 1E-9 * fI_ConveyorSpeed;
      _nCamStartPos   := _nX0 +   F_MeterToSubPixel(fPosMeter:=_fTriggerDistance, fResoSubPx:=_nResolution);
      
      // effective started position
      fDeltaDistance  := UINT64_TO_LREAL(UInt64Sub64(ULINT_TO_ULARGE(tCurrentTime), ULINT_TO_ULARGE(tTriggerFeedback_TimeStamp))) * 1E-9 * fI_ConveyorSpeed;
      _nCamStartedPos := iI_CurrentPos - F_MeterToSubPixel(fPosMeter:=fDeltaDistance, fResoSubPx:=_nResolution);
      IF _bManualStart THEN iActiveCam.CamTrigger(bOk:=bTriggerOk, nPos:=_nCamStartPos, nPosDeviation:=0, nX0:=_nX0);
      ELSE                  iActiveCam.CamTrigger(bOk:=bTriggerOk, nPos:=_nCamStartPos, nPosDeviation:=-_nCamStartedPos+_nCamStartPos, nX0:=_nX0); END_IF  (*!!!!   sign inverted*)
    ELSE
     eState           := cL_WAITFEEDBACK;
    END_IF    
    
  cL_TRIGACTIVE:   (*Trigger high*)
    eState         := cL_WAITSTOP;
    
    // calculate end timestamp of trigger (end of trigger active signal)
    tTrigger_EventTime := (tTrigger_EventTime + LREAL_TO_ULINT(_fTriggerLength * 1E6));
     
    OnTriggerCommand := nC_EL2252Cmd_INACTIVE;
    ObTrigger        := FALSE;
    
  cL_WAITSTOP:  (*Wait until trigger time has elapsed*)
    IF (tTrigger_EventTime < tCurrentTime) THEN (* StopTime elapsed *)
      eState           := cL_IDLE;
      OnTriggerCommand := nC_EL2252Cmd_INACTIVE; (*Disarm EL2252, trigger generated*)
      iActiveCam.CamTriggerDone();
    ELSE
      eState           := cL_WAITSTOP;
      IF _bUseCameraTrigger THEN
        OnTriggerCommand := nC_EL2252Cmd_ACTIVE;  (*Arm EL2252*)
      END_IF
    END_IF;

    ObTrigger        := FALSE;

  ELSE  (*Default*)
    eState           := cL_IDLE;
    ObTrigger        := FALSE;
    OnTriggerCommand := nC_EL2252Cmd_INACTIVE;
END_CASE;

OtTriggerStartTime := tTrigger_EventTime;  // set output

_tMemTriggerFeedback_TimeStampPos := tI_TriggerFeedback_TimeStampPos;

PROPERTY bManualTeach : BOOL
GET
bManualTeach := _bCamManualTeachMode;
END_GET
SET
_bCamManualTeachMode := bManualTeach;
END_SET
END_PROPERTY

(*
  A new container detected on X0.
  NOTE: a pulse only
*)
PROPERTY bStartTrig : BOOL
GET
bStartTrig := bSheetDetected;
END_GET
END_PROPERTY

(*
  A valid container detected.
*)
PROPERTY bValid : BOOL
GET
bValid := bSheetDetected AND NOT _bCamManualTeachMode AND bCamValid;  // in manual teach the ct is "present" should not be printed
END_GET
END_PROPERTY

METHOD Disable : BOOL
IF eState = cL_IDLE THEN
  iActiveCam := 0;
  Disable := TRUE;
ELSE  
  Disable := FALSE;
  LogError('disable failed: trigger busy -> reset trigger');
  Reset();
END_IF
END_METHOD

METHOD Enable : BOOL
VAR_INPUT
	iCam	                    : I_CameraTriggerDevice;
  bUseCameraTrigger         : BOOL; //Generate camera trigger
  bUseCameraTriggerFeedback : BOOL; //Use feedback as trigger?
END_VAR
IF iCam = 0 THEN
  Enable := FALSE;
  LogError('setCam failed: invalid reference');
ELSIF eState <> cL_IDLE THEN
  Enable := FALSE;
  LogError('enable failed: trigger busy');
ELSE
  iActiveCam := iCam;
  Enable     := TRUE;

  // save constant settings
  _bUseCameraTrigger := bUseCameraTrigger;
  _bUseCameraTriggerFeedback := bUseCameraTriggerFeedback;
END_IF;
END_METHOD

METHOD Init
VAR_INPUT
  nResolution                   : INT := 1;        (*Printhead Resolution [e.g. 600] x Subpixel Resolution [e.g. 32]*)
  bUsePositionTrigger           : BOOL;            (*FALSE: Calculate time with speed and position distance@sensor event*)
END_VAR
(*zero divisions*)
IF nResolution = 0 THEN 
  bInitOk :=FALSE;
  RETURN; 
END_IF;

_nResolution:=nResolution;
_bUsePositionTrigger :=bUsePositionTrigger;


bInitOk :=TRUE;
END_METHOD

(*
  Log timestamp difference (if verbose active).
  t1-t2 
*)
METHOD LogTsDiff : BOOL
VAR_INPUT
  aIdent : STRING;
  t1 : T_DCTIME64;
  t2 : T_DCTIME64;
END_VAR
IF _bVerbose THEN
  LogLvl(Lvl:=E_LogSeverity.Debug, Msg:=
       F_Concat7(aIdent, 
                 't1: ', TO_STRING(t1), 
                 ' t2: ', TO_STRING(t2), 
                 ' t1-t2 [ms]: ', TO_STRING((TO_LREAL(t1)-TO_LREAL(t2))*1E-6)
       )
  );
END_IF
END_METHOD

(*
  Detected start position X0 (absolute) in [SubPx].
*)
PROPERTY nStartPositionX0 : DINT
GET
nStartPositionX0 := _nX0;
END_GET
END_PROPERTY

METHOD Reset
VAR_INPUT
END_VAR
eState              := cL_IDLE;      // reset state
OtTriggerStartTime  := F_GetCurDcTaskTime64();  // now
ObTrigger           := FALSE;        // set output = 0
OnTriggerCommand    := nC_EL2252Cmd_ACTIVE;    // activate command
bInhibitTrigger := FALSE;
END_METHOD

METHOD SetSubstrateLength
VAR_INPUT
  fSubstrateLength : LREAL;
END_VAR
IF NOT bInitOk THEN RETURN;END_IF;

(*Added 10 mm margin for substrate length in case of print quality strips at the end of sheet in case of start with edge*)
_fSubstrateLength := fSubstrateLength + fC_SheetLengthMargin;
_nSubstrateLength := F_MeterToSubPixel(fPosMeter:=_fSubstrateLength, fResoSubPx:=_nResolution);
END_METHOD

END_FUNCTION_BLOCK

// ---- POUs/Print/Camera/FB_MarkCamera.TcPOU
(*
  Mark camera system
  2 mark sensors detect sheet marks.   
*)
FUNCTION_BLOCK FB_MarkCamera EXTENDS FB_CameraBase 

VAR_INPUT
  IbSensorState       AT%I* : ARRAY [1..cNbSensors] OF BOOL;        (*Mark sensor state*)
  ItTimeStampPos      AT%I* : ARRAY [1..cNbSensors] OF T_DCTIME64;  (*TimeStamp Pos_Edge @EL1252*)
  ItTimeStampNeg      AT%I* : ARRAY [1..cNbSensors] OF T_DCTIME64;  (*TimeStamp Neg_Edge @EL1252*)

  IfConveyorSpeed           : LREAL;      (*Actual speed of conveyor [m/s]*)
  IfMasterPosition          : LREAL;      (*Master position [µm]*)
END_VAR

VAR
  nCounter                  : UDINT;

  _fSensorDistance          : REAL := 1.0;    (*Distance between the two sensors [m]*)
  _fMarkPositionX           : REAL := 0.010;  (*Distance sheet edge to mark position [m]*)
  _fMarkSizeX               : REAL;           (*Mark size X [mm]*)
  _fMarkSizeY               : REAL;           (*Mark size Y [mm]*)

  tSensorRisingEdge         : ARRAY [1..cNbSensors] OF T_DCTIME64;
  tSensorFallingEdge        : ARRAY [1..cNbSensors] OF T_DCTIME64;
  bMemSensorState           : ARRAY [1..cNbSensors] OF BOOL;       (*Mem mark sensor state*)
  bInhibSensor              : ARRAY [1..cNbSensors] OF BOOL;       (*Inhibit sensor signals, TRUE=inhibit*)
  bSensorStateOK            : ARRAY [1..cNbSensors] OF BOOL;       (*Mark sensor state ok*)
  fSensorDuration           : ARRAY [1..cNbSensors] OF REAL;       (*Sensor signal duration [ns]*)
  fSensorLength             : ARRAY [1..cNbSensors] OF REAL;       (*Sensor signal length [mm]*)
  fS1S2EdgeDistance         : REAL;       (*Edge distance between sensors [mm]*)
  fLateralOffset            : REAL;       (*Lateral offset [mm]*)
  fMemMasterPosition        : LREAL;      (*Mem master position [µm]*)
  bStopCondition            : BOOL;       (*Condition for stop trigger*)
END_VAR

VAR CONSTANT                
  cNbSensors                : UDINT := 2; (*Number of mark sensors*)
END_VAR

IF NOT _bInitialized THEN RETURN; END_IF

(*check parameter*)
IF _fSensorDistance = 0 THEN
	_fSensorDistance := 1.0;
END_IF;

FOR nCounter := 1 TO cNbSensors DO
  (* -------- Detection of rising edge on sensor --------*)
  IF IbSensorState[nCounter] AND NOT bMemSensorState[nCounter] AND NOT bInhibSensor[nCounter] THEN
    tSensorRisingEdge[nCounter] := ItTimeStampPos[nCounter];
    fMemMasterPosition          := IfMasterPosition;
  END_IF;
  
  (* -------- Detection of falling edge --------*)
  IF NOT IbSensorState[nCounter] AND bMemSensorState[nCounter] AND NOT bInhibSensor[nCounter] THEN
    tSensorFallingEdge[nCounter] := ItTimeStampNeg[nCounter];
    fSensorDuration   [nCounter] := LREAL_TO_REAL(ULINT_TO_LREAL(tSensorFallingEdge[nCounter]) - ULINT_TO_LREAL(tSensorRisingEdge[nCounter]));		(* Calculate how long the signal was ON *)
    fSensorLength     [nCounter] := LREAL_TO_REAL(fSensorDuration[nCounter] * IfConveyorSpeed / 1_000_000_000);			(* Calculate the equivalence in mm *)
    bSensorStateOK    [nCounter] := TRUE;   (* now the function can continue to Angle & Offset calculation *)
    bInhibSensor      [nCounter] := TRUE;
  END_IF;
  
  bMemSensorState[nCounter] := IbSensorState[nCounter];			(* Memorization of the sensor1 state for next cycle *)
END_FOR

(* ------------ ANGLE & OFFSET CALCULATION ----------------- *)
IF bSensorStateOK[1] AND bSensorStateOK[2] THEN
  fS1S2EdgeDistance := LREAL_TO_REAL(ULINT_TO_LREAL(tSensorRisingEdge[1] - tSensorRisingEdge[2]) / 1_000_000 * IfConveyorSpeed);	(* Calculate the difference in mm between S1 and S2 trigger *)

  fLateralOffset := (_fMarkSizeY / _fMarkSizeX) * (fSensorLength[1] - fSensorLength[2]) / 2;  (* Evaluation of the offset for each mark *)

  IF _iCameraSink <> 0 THEN
    (*Mark1*)
    stCamPoint.x_ref := F_MeterToSubPixelReal( _fMarkPositionX                                      (*[m]*)
                                              , UDINT_TO_LREAL(_nPrintUnitResolution));             (*Result should be in pixels*)
    stCamPoint.y_ref := F_MeterToSubPixelReal( (_fSubstrateWidth / 2) - (_fSensorDistance / 2)       (*[m]*)
                                              , UDINT_TO_LREAL(_nPrintUnitResolution));             (*Result should be in pixels*)
    stCamPoint.dx    := 0;
    stCamPoint.dy    := F_MeterToSubPixelReal( fLateralOffset * 0.001                              (*[mm] => [m]*)
                                              , UDINT_TO_LREAL(_nPrintUnitResolution));             (*Result should be in pixels*)
    stCamPoint.valid := TRUE;
    
    _iCameraSink.AddCamPoint(stCamPoint);
    _nRxCamPoints := _nRxCamPoints + 1 ;
  
    (*Mark2*)
    stCamPoint.x_ref := F_MeterToSubPixelReal( _fMarkPositionX                                      (*[m]*)
                                             , UDINT_TO_LREAL(_nPrintUnitResolution));             (*Result should be in pixels*)
    stCamPoint.y_ref := F_MeterToSubPixelReal( (_fSubstrateWidth / 2) - (_fSensorDistance / 2) + _fSensorDistance  (*[m]*)
                                             , UDINT_TO_LREAL(_nPrintUnitResolution));             (*Result should be in pixels*)
    stCamPoint.dx    := F_MeterToSubPixelReal( fS1S2EdgeDistance * 0.001                           (*[mm] => [m]*)
                                             , UDINT_TO_LREAL(_nPrintUnitResolution));             (*Result should be in pixels*)
    stCamPoint.dy    := F_MeterToSubPixelReal( fLateralOffset * 0.001                              (*[mm] => [m]*)
                                             , UDINT_TO_LREAL(_nPrintUnitResolution));             (*Result should be in pixels*)
    stCamPoint.valid := TRUE;
    
    _iCameraSink.AddCamPoint(stCamPoint);
    _nRxCamPoints := _nRxCamPoints + 1;
  END_IF;

	bSensorStateOK[1]  := FALSE;
	bSensorStateOK[2]  := FALSE;
END_IF;


(*------------ start and stop signal treatment ------------*)
(*generate stop trigger*)
bStopCondition := (IfMasterPosition >= (fMemMasterPosition + (_fSubstrateLength * 1_000_000)));

IF bStopCondition AND (bInhibSensor[1] OR bInhibSensor[2]) THEN
  bInhibSensor[1] := FALSE;
  bInhibSensor[2] := FALSE;
END_IF;

// TODO: 'implement PUC messages eCPr_PrintMarkError1&2'

{attribute 'monitoring':='call'}
PROPERTY eCameraMode : E_CameraMode
GET
eCameraMode := _eCameraMode;
IF _eCameraMode = E_CameraMode.Auto THEN
  eCameraMode := E_CameraMode.XYR;
END_IF
END_GET
END_PROPERTY

PROPERTY eDeviceType : E_CameraDevice
GET
eDeviceType := E_CameraDevice.PrintMark;
END_GET
END_PROPERTY

PROPERTY fMarkPositionX : REAL
SET
_fMarkPositionX := fMarkPositionX;
END_SET
END_PROPERTY

PROPERTY fMarkSizeX : REAL
SET
_fMarkSizeX := fMarkSizeX;
END_SET
END_PROPERTY

PROPERTY fMarkSizeY : REAL
SET
_fMarkSizeY := fMarkSizeY;
END_SET
END_PROPERTY

PROPERTY fSensorDistance : REAL
SET
_fSensorDistance := fSensorDistance;
END_SET
END_PROPERTY

METHOD GetCamStatus : BOOL
VAR_OUTPUT
  bConnectionOK  : BOOL;    // Camera connected
  bTeachOk       : BOOL;    // Teach successful
  nTeachedPoints : UDINT;   // Teached points for this job
  nScannedPoints : UDINT;   // Scanned points on current sheet
  bCamStarted    : BOOL;    // Camera trigger is active, cam started
  bCamDone       : BOOL;    // Camera finished on last CT
  bErrors        : ARRAY[1..GVL_Camera.nC_NbCamErrors] OF BOOL;  // generic error flag list
END_VAR
bConnectionOK  := TRUE;
bTeachOk       := TRUE; // NO teach availabe
nTeachedPoints := 2;    // 2 marks only
nScannedPoints := _nRxCamPoints;
bCamStarted    := _bCamTriggerStarted;
bCamDone       := _bCamTriggerDone;

GetCamStatus := bConnectionOK AND bTeachOk;   // camera ready
END_METHOD

METHOD InitMarkCamera
VAR_INPUT
  nPrintUnitResolution         : UDINT;    (*printhead pixel resolution [dpi]*)
  nPrintUnitSubPx              : UDINT;    (*print unit subPixel resolution [SubPx]*)
  iCameraTrigger               : I_CameraTrigger;
END_VAR
SUPER^.Init( nPrintUnitResolution      := nPrintUnitResolution
           , nPrintUnitSubPx           := nPrintUnitSubPx
           , iCameraTrigger            := iCameraTrigger
           , bUseCameraTrigger         := FALSE
           , bUseCameraTriggerFeedback := FALSE);

_bInitialized := TRUE;
END_METHOD

(*
  Set mode to camera.
  :return: TRUE if success
*)
METHOD setCameraMode : BOOL
VAR_INPUT
  eCameraMode : E_CameraMode;
END_VAR
IF eCameraMode = E_CameraMode.NoCorrection OR  // supported modi
   eCameraMode = E_CameraMode.XYR THEN
   
  _eCameraMode := eCameraMode;  // set desired mode
  setCameraMode := TRUE;
ELSE
  LogError(F_Concat3('Camera mode=', TO_STRING(eCameraMode), ' not supported by camera'));
  _eCameraMode := E_CameraMode.NoCorrection;
END_IF
END_METHOD

{attribute 'monitoring':='variable'}
PROPERTY sName : STRING
GET
sName := 'Printmarks';
END_GET
END_PROPERTY

END_FUNCTION_BLOCK

// ---- POUs/Print/Camera/FB_SystronCamera.TcPOU
(*
  Systron camera system
  Provides callback function (rx_callback) for received TcpIp messages.   
*)
FUNCTION_BLOCK FB_SystronCamera EXTENDS FB_CameraTcpIp

VAR
  stCameraResult            : ARRAY [1..cNbCameras] OF ST_CAMERA_RESULT;

  nNbTrigger                : INT;
END_VAR

VAR CONSTANT                
  cNbCameras                : UDINT := 2;                (*Number of Systron cameras*)

  cErrorString              : T_MaxString := '<Error(';
  cStartString              : T_MaxString := '<position(';
  cEndingString             : T_MaxString := ');';

  cCameraMinXY              : REAL := -20.0;  (*[mm]*)
  cCameraMaxXY              : REAL := +20.0;  (*[mm]*)
END_VAR

(*Simulation*)
IF _bSimulate THEN
  CreateSimCamPoints();
END_IF

(*
  Simulate camera data
*)
METHOD CreateSimCamPoints : BOOL
VAR_INST
  fbTonTimer    : TON;    (*Send timer*)
  nCounter      : UDINT;  (*Loop counter*)
END_VAR
(*Test points*)
stCameraResult[1].x_ref :=   54;  (*[mm]*)
stCameraResult[1].y_ref := 1003;  (*[mm]*)
stCameraResult[1].valid := TRUE;
stCameraResult[2].x_ref :=   46;  (*[mm]*)
stCameraResult[2].y_ref :=  376;  (*[mm]*)
stCameraResult[2].valid := TRUE;

(*Points are send every 15s*)
fbTonTimer(IN := NOT fbTonTimer.Q, PT := T#15S);
IF fbTonTimer.Q THEN
  FOR nCounter := 1 TO 2 DO
    stCamPoint.x_ref := F_MeterToSubPixelReal( stCameraResult[nCounter].x_ref * 0.001      (*[mm] => [m]*)
                                             , UDINT_TO_LREAL(_nPrintUnitResolution));     (*Result should be in pixels*)
    stCamPoint.y_ref := F_MeterToSubPixelReal( stCameraResult[nCounter].y_ref * 0.001      (*[m]*)
                                             , UDINT_TO_LREAL(_nPrintUnitResolution));     (*Result should be in pixels*)
    stCamPoint.dx    := F_MeterToSubPixelReal( 0.100 * UDINT_TO_REAL(nCounter) * 0.001     (*[mm] => [m]*)
                                            , UDINT_TO_LREAL(_nPrintUnitResolution));     (*Result should be in pixels*)
    stCamPoint.dy    := F_MeterToSubPixelReal( 0.200 * UDINT_TO_REAL(nCounter) * 0.001     (*[mm] => [m]*)
                                            , UDINT_TO_LREAL(_nPrintUnitResolution));     (*Result should be in pixels*)
  
    _iCameraSink.AddCamPoint(stCamPoint);
  END_FOR  
END_IF
END_METHOD

{attribute 'monitoring':='call'}
PROPERTY eCameraMode : E_CameraMode
GET
eCameraMode := _eCameraMode;
IF _eCameraMode = E_CameraMode.Auto THEN
  eCameraMode := E_CameraMode.XYR;
END_IF
END_GET
END_PROPERTY

PROPERTY eDeviceType : E_CameraDevice
GET
eDeviceType := E_CameraDevice.PrintMark;
END_GET
END_PROPERTY

METHOD GetCamStatus : BOOL
VAR_OUTPUT
  bConnectionOK  : BOOL;    // Camera connected
  bTeachOk       : BOOL;    // Teach successful
  nTeachedPoints : UDINT;   // Teached points for this job
  nScannedPoints : UDINT;   // Scanned points on current sheet
  bCamStarted    : BOOL;    // Camera trigger is active, cam started
  bCamDone       : BOOL;    // Camera finished on last CT
  bErrors        : ARRAY[1..GVL_Camera.nC_NbCamErrors] OF BOOL;  // generic error flag list
END_VAR
bConnectionOK  := NOT bConnectionErr OR bSimulate;
bTeachOk       := TRUE; //NO teach availabe (teached by a specific sheet from machine)
nTeachedPoints := 0;
nScannedPoints := 0;
bCamStarted    := _bCamTriggerStarted;
bCamDone       := _bCamTriggerDone;

GetCamStatus := bConnectionOK;
END_METHOD

METHOD rx_callback
VAR_INPUT
	sMessage	: CalmarCompTcpIp.ST_TcpMsg;
END_VAR

VAR
  sAnalyzeLastMessage    : T_MaxString;          (*telegram string*)

  nCounter               : UDINT;
  nFindIndex             : INT;
END_VAR
SUPER^.rx_callback(sMessage := sMessage);

sAnalyzeLastMessage := sLastMessage;

nFindIndex := FIND(sAnalyzeLastMessage, cErrorString);
IF nFindIndex > 0 THEN
  (*Error received*)
  sLastErrorMessage := (DELETE(sAnalyzeLastMessage, (nFindIndex + LEN(cErrorString) - 1), 1));

  (*Extract error message*)
  nFindIndex := FIND(sLastErrorMessage, cEndingString);
  IF nFindIndex > 0 THEN
    sLastErrorMessage := (DELETE(sLastErrorMessage, LEN(sLastErrorMessage) - nFindIndex, nFindIndex));
  END_IF;
ELSE
  (*Search for start string*)
  nFindIndex := FIND(sAnalyzeLastMessage, cStartString);
  IF nFindIndex > 0 THEN
    (*Search string found => remove string to generate index*)
    sAnalyzeLastMessage := (DELETE(sAnalyzeLastMessage, (nFindIndex + LEN(cStartString) - 1), 1));

    (*Search for trigger number*)
    nFindIndex := FIND(sAnalyzeLastMessage, ',');
    IF nFindIndex > 0 THEN
      nNbTrigger := STRING_TO_INT(LEFT(sAnalyzeLastMessage, (nFindIndex - 1)));

      sAnalyzeLastMessage := (DELETE(sAnalyzeLastMessage, nFindIndex, 1));
    END_IF;

    (*Search for rx, ry, v, x and y*)
    FOR nCounter := 1 TO cNbCameras DO
      stCameraResult[nCounter].valid := TRUE;

      (*rx*)
      nFindIndex := FIND(sAnalyzeLastMessage, ',');
      IF nFindIndex > 0 THEN
        stCameraResult[nCounter].x_ref := STRING_TO_REAL(LEFT(sAnalyzeLastMessage, (nFindIndex - 1)));

        IF    (stCameraResult[nCounter].x_ref < cCameraMinXY)
           OR (stCameraResult[nCounter].x_ref > cCameraMaxXY)
        THEN
          stCameraResult[nCounter].valid := FALSE;
        END_IF;

        sAnalyzeLastMessage := (DELETE(sAnalyzeLastMessage, nFindIndex, 1));
      ELSE
        stCameraResult[nCounter].valid := FALSE;
      END_IF;
      (*ry*)
      nFindIndex := FIND(sAnalyzeLastMessage, ',');
      IF nFindIndex > 0 THEN
        stCameraResult[nCounter].y_ref := STRING_TO_REAL(LEFT(sAnalyzeLastMessage, (nFindIndex - 1)));

        IF    (stCameraResult[nCounter].y_ref < cCameraMinXY)
           OR (stCameraResult[nCounter].y_ref > cCameraMaxXY)
        THEN
          stCameraResult[nCounter].valid := FALSE;
        END_IF;

        sAnalyzeLastMessage := (DELETE(sAnalyzeLastMessage, nFindIndex, 1));
      ELSE
        stCameraResult[nCounter].valid := FALSE;
      END_IF;
      (*v*)
      nFindIndex := FIND(sAnalyzeLastMessage, ',');
      IF nFindIndex > 0 THEN
        IF FIND(LEFT(sAnalyzeLastMessage, (nFindIndex - 1)), 'True') > 0 THEN
          stCameraResult[nCounter].valid := TRUE;
        ELSE
          stCameraResult[nCounter].valid := FALSE;
        END_IF;

        sAnalyzeLastMessage := (DELETE(sAnalyzeLastMessage, nFindIndex, 1));
      ELSE
        stCameraResult[nCounter].valid := FALSE;
      END_IF;
      (*x*)
      nFindIndex := FIND(sAnalyzeLastMessage, ',');
      IF nFindIndex > 0 THEN
        stCameraResult[nCounter].x := STRING_TO_REAL(LEFT(sAnalyzeLastMessage, (nFindIndex - 1)));

        IF    (stCameraResult[nCounter].x < cCameraMinXY)
           OR (stCameraResult[nCounter].x > cCameraMaxXY)
        THEN
          stCameraResult[nCounter].valid := FALSE;
        END_IF;

        sAnalyzeLastMessage := (DELETE(sAnalyzeLastMessage, nFindIndex, 1));
      ELSE
        stCameraResult[nCounter].valid := FALSE;
      END_IF;
      (*y*)
      nFindIndex := FIND(sAnalyzeLastMessage, ',');
      IF nFindIndex > 0 THEN
        stCameraResult[nCounter].y := STRING_TO_REAL(LEFT(sAnalyzeLastMessage, (nFindIndex - 1)));

        IF    (stCameraResult[nCounter].y < cCameraMinXY)
           OR (stCameraResult[nCounter].y > cCameraMaxXY)
        THEN
          stCameraResult[nCounter].valid := FALSE;
        END_IF;

        sAnalyzeLastMessage := (DELETE(sAnalyzeLastMessage, nFindIndex, 1));
      ELSE
        nFindIndex := FIND(sAnalyzeLastMessage, ')');
        IF nFindIndex > 0 THEN
          stCameraResult[nCounter].y := STRING_TO_REAL(LEFT(sAnalyzeLastMessage, (nFindIndex - 1)));

          IF    (stCameraResult[nCounter].y < cCameraMinXY)
             OR (stCameraResult[nCounter].y > cCameraMaxXY)
          THEN
            stCameraResult[nCounter].valid := FALSE;
          END_IF;

          sAnalyzeLastMessage := (DELETE(sAnalyzeLastMessage, nFindIndex, 1));
        ELSE
          stCameraResult[nCounter].valid := FALSE;
        END_IF;
      END_IF;
    END_FOR;
  ELSE
    (*Search string not found*)
    FOR nCounter := 1 TO cNbCameras DO
      stCameraResult[nCounter].valid := FALSE;
    END_FOR;
  END_IF;
END_IF;

IF _iCameraSink <> 0 THEN
  FOR nCounter := 1 TO cNbCameras DO
    stCamPoint.x_ref := F_MeterToSubPixelReal( stCameraResult[nCounter].x_ref * 0.001              (*[mm] => [m]*)
                                         , UDINT_TO_LREAL(_nPrintUnitResolution));             (*Result should be in pixels*)
    stCamPoint.y_ref := F_MeterToSubPixelReal( stCameraResult[nCounter].y_ref * 0.001              (*[m]*)
                                         , UDINT_TO_LREAL(_nPrintUnitResolution));             (*Result should be in pixels*)
    stCamPoint.dx    := F_MeterToSubPixelReal( (stCameraResult[nCounter].x_ref - stCameraResult[nCounter].x) * 0.001  (*[mm] => [m]*)
                                         , UDINT_TO_LREAL(_nPrintUnitResolution));             (*Result should be in pixels*)
    stCamPoint.dy    := F_MeterToSubPixelReal( (stCameraResult[nCounter].y_ref - stCameraResult[nCounter].y) * 0.001  (*[mm] => [m]*)
                                         , UDINT_TO_LREAL(_nPrintUnitResolution));             (*Result should be in pixels*)

    _iCameraSink.AddCamPoint(stCamPoint);
  END_FOR
END_IF;

bMsgReceived := FALSE;
END_METHOD

(*
  Set mode to camera.
  :return: TRUE if success
*)
METHOD setCameraMode : BOOL
VAR_INPUT
  eCameraMode : E_CameraMode;
END_VAR
IF eCameraMode = E_CameraMode.NoCorrection OR  // supported modi
   eCameraMode = E_CameraMode.XYR THEN
 
  _eCameraMode := eCameraMode;  // set desired mode
  setCameraMode := TRUE;
ELSE
  LogError(F_Concat3('Camera mode=', TO_STRING(eCameraMode), ' not supported by camera'));
  _eCameraMode := E_CameraMode.NoCorrection;
END_IF
END_METHOD

{attribute 'monitoring':='variable'}
PROPERTY sName : STRING
GET
sName := 'Systron';
END_GET
END_PROPERTY

END_FUNCTION_BLOCK

// ---- POUs/Print/Camera/FB_TcpIpComm.TcPOU
FUNCTION_BLOCK FB_TcpIpComm EXTENDS T_NamedBase IMPLEMENTS I_BootService
VAR_INPUT
END_VAR
VAR_OUTPUT
END_VAR
VAR
  // boot service
  _bStarting       : BOOL := TRUE;
  _tStartDelay     : ARRAY[1..nMaxTcpIpClients] OF TIME;
  fbTonStartDelay  : ARRAY[1..nMaxTcpIpClients] OF TON;
  
  // TcpIp clients list
  sSrvNetId        : T_AmsNetID := '';           (* AmsId of tcpip server.exe, default: empty string. *)
  fbCloseAll       : FB_SocketCloseAll;          (* close all opened sockets *)
  
  fbTcpClients     : ARRAY[1..nMaxTcpIpClients] OF FB_TcpClient;
  pActiveClients   : ARRAY[1..nMaxTcpIpClients] OF POINTER TO FB_TcpClient;
  nActiveTcpClients: UINT;    // active/registered clients¨
  
  nCtr  : UINT;
END_VAR
VAR CONSTANT
  nMaxTcpIpClients      : UINT := 4;
END_VAR

IF _bStarting THEN RETURN; END_IF

// call all active clients
FOR nCtr:=1 TO nActiveTcpClients DO
  fbTonStartDelay[nCtr](IN := TRUE, PT := _tStartDelay[nCtr]);
  IF fbTonStartDelay[nCtr].Q THEN
    fbTcpClients[nCtr](
      //bEnable := .....
      //bConnected => 
    );
  END_IF
END_FOR

PROPERTY bStarting : BOOL
GET
// return booint satus to boot service
bStarting := _bStarting;
END_GET
END_PROPERTY

METHOD closeAllSockets : BOOL
VAR_INST
  bClosing  : BOOL;
END_VAR
(* close all opened/created sockets *)
IF NOT bClosing THEN fbCloseAll( sSrvNetId := sSrvNetId, bExecute:= FALSE ); bClosing := TRUE; END_IF  // be sure to call it once with FALSE

fbCloseAll( sSrvNetId := sSrvNetId, bExecute:= bClosing );
IF NOT fbCloseAll.bBusy THEN
  // done
  //IF fbCloseAll.bError THEN LogError(F_Concat2('CloseAllSockets error=', F_GetAdsErrDescription(lErrCode:=fbCloseAll.nErrId))); 
  //ELSE                      LogInfo('CloseAllSockets done.'); END_IF
  bClosing := FALSE;
END_IF

// return busy
closeAllSockets := fbCloseAll.bBusy;
END_METHOD

METHOD registerTcpIpClient : POINTER TO FB_TcpClient
VAR_INPUT
  sRemoteHost   : ST_SockAddr;
  iHandler      : I_TcpIp_RxMsgHandler;
  tStartDelay   : TIME;
END_VAR

VAR
  pTcpIpClient  : POINTER TO FB_TcpClient;
END_VAR
IF nActiveTcpClients >= nMaxTcpIpClients THEN
  LogError('No free TcpIp client, ignore registerTcpIpClient');
END_IF

nActiveTcpClients := nActiveTcpClients + 1;

// config
fbTcpClients[nActiveTcpClients].sRemoteHost := sRemoteHost.sAddr;
fbTcpClients[nActiveTcpClients].nRemotePort := sRemoteHost.nPort;
_tStartDelay[nActiveTcpClients]             := tStartDelay;

// init
fbTcpClients[nActiveTcpClients].init(
  tReconnect := T#100MS,
  tRxPolling := T#1MS,
  //cMsgTermination := cMSG_TERMINATION_ZERO
);
// start
fbTcpClients[nActiveTcpClients].bEnable := TRUE;
fbTcpClients[nActiveTcpClients].register_RxMsgHandler(bAdd:=TRUE, iHandler);

// return client handle (pointer = full access)
pActiveClients[nActiveTcpClients] := ADR(fbTcpClients[nActiveTcpClients]);
registerTcpIpClient := ADR(fbTcpClients[nActiveTcpClients]);
END_METHOD

METHOD start : BOOL
// called by system boot services, 'regBootService' needed
IF NOT closeAllSockets() THEN
  // done 
  _bStarting := FALSE;  // we are done
END_IF

start := _bStarting;
END_METHOD

END_FUNCTION_BLOCK

// ---- POUs/Print/Camera/F_DeformationPointAcc_ToString.TcPOU
FUNCTION F_DeformationPointAcc_ToString : T_MaxString
VAR_INPUT
  sPointAcc : ST_DeformationPointAccurate;
END_VAR

F_DeformationPointAcc_ToString := F_Concat4(
  F_Concat4('idx: ', TO_STRING(sPointAcc.index), ' v: ', SEL(sPointAcc.valid>0, '0', '1')),
  F_Concat5(' c/r(', TO_STRING(sPointAcc.col), '/', TO_STRING(sPointAcc.row),')'),
  F_Concat4(' x_ref: ' , LREAL_TO_FMTSTR(sPointAcc.x_ref, 4, TRUE),' y_ref: ', LREAL_TO_FMTSTR(sPointAcc.y_ref, 4, TRUE)),
  F_Concat4(' dx: ' , LREAL_TO_FMTSTR(sPointAcc.dx, 4, TRUE),' dy: ', LREAL_TO_FMTSTR(sPointAcc.dy, 4, TRUE))
);

END_FUNCTION

// ---- POUs/Print/Camera/F_CamPoint_ToString.TcPOU
FUNCTION F_CamPoint_ToString : T_MaxString
VAR_INPUT
  sPoint : ST_CameraPoint;
END_VAR

F_CamPoint_ToString := F_Concat3(
  F_Concat4('id: ', TO_STRING(sPoint.id), ' v: ', SEL(sPoint.valid>0, '0', '1')),
  F_Concat4(' x_ref: ' , TO_STRING(sPoint.x_ref),' y_ref: ', TO_STRING(sPoint.y_ref)),
  F_Concat4(' dx: ' , TO_STRING(sPoint.x),' dy: ', TO_STRING(sPoint.y))
);

END_FUNCTION

// ---- POUs/Print/Camera/LineCamera/FB_LineCamera.TcPOU
(*
  QualiVision line camera system
  Provides callback function (rx_callback) for received TcpIp messages.   
*)
FUNCTION_BLOCK FB_LineCamera EXTENDS FB_CameraTcpIp IMPLEMENTS I_Sim

VAR_INPUT
  InTempActValueScanner   AT%I* : INT;    (*Actual value temperature camera [0.1 C]*)
  InTempActValuePrintUnit       : INT;    (*Actual value temperature pu [0.1 C]*)
  IfSpeed                       : LREAL;  (*Actual speed [m/s]*)
END_VAR

VAR
  _fCameraWidthNormal       : LREAL;       (*cW: Camera width [m]*)
  _nCameraWidth             : DINT;        (*Camera width [px]*)
  _fCameraMechOffsetTC      : LREAL;       (*Camera mechanical offset at calibration temp [mm]*)
  _fMechOffsetCameraToPU    : LREAL;       (*Camera mechanical offset to PrintUnit [mm]*)
  _fPrintUnitMechOffsetTC   : LREAL;       (*PrintUnit mechanical offset at calibration temp [mm]*)
  _nPrintUnitWidthNormal    : UDINT;       (*Print unit width [px] native*)
  _fPrintUnitWidthTC        : LREAL;       (*pWc: Print unit width [m]*)
  _fPrintUnitCalTemp        : LREAL;       (*calibration temperature for the PrintUnit*)

  fCameraWidthTC            : LREAL;       (*cWc: Camera width [m] at specific calibration temperature*)
  fCameraTemp               : LREAL;       (*Camera actual temp [°C]*)
  fCameraDeltaTempFactor    : LREAL;       (*Factor for distance calculation at delta temp*)
  fCameraRealResolution     : LREAL;       (*real resolution (with the actual temperature) from the line camera in y direction*)
  fCameraMechOffsetTAct     : LREAL;       (*Camera mechanical offset at actual temp [mm]*)
  fCameraCenterOffsetTAct   : LREAL;       (*Camera center offset at actual temp [mm]*)
  
  fPrintUnitTemp            : LREAL;       (*PrintUnit actual temp [°C]*)
  fPrintUnitDeltaTempFactor : LREAL;       (*Factor for distance calculation at delta temp*)
  fPrintUnitMechOffsetTAct  : LREAL;       (*PrintUnit mechanical offset at actual temp [mm]*)
  fPrintUnitWidthTAct       : LREAL;       (*PrintUnit width at actual temp [mm]*)
  fPrintUnitWidthDiff       : LREAL;       (*PrintUnit width difference at actual temp [mm]*)
  fPrintUnitCenterOffsetTAct: LREAL;       (*PrintUnit center offset at actual temp [mm]*)

  fCameraDelay              : LREAL;      (*camera start delay from frame grabber (300dpi vs 600dpi phase sync.) in [m]*)            
  
  nNbVersion                : INT;
  sModus                    : T_MaxString;
  nSector                   : DINT;
  nNbMarks                  : UDINT;
  _bTeachOk                 : BOOL;
  nNbMarksTeach             : UDINT;
  nNbMarksScanned           : UDINT;
  nNbSectorTeach            : DINT;
  sTeach                    : T_MaxString;      // last teach message (255 chars only), for VISU only
  sCameraPoints             : ARRAY [1..GVL_Camera.cMaxNbMarks] OF ST_CameraPoint;   // camera points list of received 'A' frames, also used for 'T' at job start
  sTeachPoints              : ARRAY [1..GVL_Camera.cMaxNbMarks] OF ST_TeachPoint;    // teached points
  nNumPointsPerSectorT      : ARRAY [1..GVL_Camera.cMaxNbSectors] OF DINT;           // number of marks in theach in frame x
  nNumPointsPerSectorA      : ARRAY [1..GVL_Camera.cMaxNbSectors] OF DINT;           // number of marks received in frame x
  nNumFrames                : UDINT;                                      // number of camera frames for job
  
  // Messages
  fbMsg_NotEnoughTeachPoints  : FB_MESSAGE;
  bNotEnoughTeachPoints : BOOL;
  bNotAllFramesContainTeachPoints : BOOL;
  bInvalidTeachPointsReceived : BOOL;
  
  // debug ------------------------
  _bVerbose                 : BOOL;   // Enable verbose mode (log more debug information
  // camera timing
  // - loop test (PLC->QR->PLC)
  _bTestTx                  : BOOL; // send a message (loop time test) from VISU button
  _tTimeTx, _tTimeRx        : T_DCTIME64;
  _sTimeElapsed             : STRING;
  _tTimeTrigger             : T_DCTIME64;
  _nTimeFrameIdx_CamMsg     : UDINT := 1;
  _tTimeFrames_CamMsg       : ARRAY[0..nC_MaxRxTimingEntries] OF T_DCTIME64;   // TimeStamp of cam messages
  _tTimeFramesMs_CamMsg     : ARRAY[0..nC_MaxRxTimingEntries] OF LREAL;        // elapsed times of each frame since trigger
  _tTimeFrames_TestMsg      : ARRAY[0..nC_MaxRxTimingEntries] OF T_DCTIME64;   // TimeStamp of test messages
  _tTimeFramesMs_TestMsg    : ARRAY[0..nC_MaxRxTimingEntries] OF LREAL;        // elapsed time of each frame since trigger 
  // tcp camera simulation
  _nSimMode                 : UDINT := 0; // 0=generate points in plc, 1=use ext. cam simulation script, 2=send rx_callback messages directly
  _sSimCamPoints            : ARRAY [1..GVL_Camera.cMaxNbMarks] OF ST_DeformationPointAccurate;
  _nSimCamFrameDepth        : UDINT := 2048;   // distance of cam frames (point pitch in x in [px])
  _nSimCamMarksPerFrame     : UDINT := 6;  
  _bSimCamPointValid        : BOOL := TRUE;
  _aCamSimScriptPath        : T_MaxString;
  fbScriptCamSim            : FB_ScriptLauncher;    // external cam simulation script
  _rfTrigSim                : RF_TRIG;
//  _tStartSim                : TON;
  // ---- NOTE: vars accesses by CameraSimulation script, edit on both sides
  nScriptPID                : UDINT;
  nFrameNr                  : UDINT;
  // -----
END_VAR                     

VAR CONSTANT
  // protocol
  cErrorString              : T_MaxString := '<Error(';  (*not used yet*)
  cStartString              : T_MaxString := '<position(';
  cEndingString             : T_MaxString := ');';
  cProtoVersion_100         : INT := 100;               // initial protocol version
  cProtoVersion_110         : INT := 110;               // protocol extension +sector indication in T and A +end sector indication
  cIdxFirstSector           : UDINT := 1;
  
  // camera
  cCameraMinXY              : DINT := 0;       (*[px/4800dpi]*)
  cCameraMaxXY              : DINT := 205_000; (*[px/4800dpi]*)
  cCameraResolution         : LREAL := 300;     (*Camera pixel resolution [dpi]*)
  cCameraResolutionSubpixel : LREAL :=  16;     (*Subpixel point resolution [SubPx] -> 4800dpi*)
  cCameraTempCoefficient    : LREAL := 23.1E-6; (*thermal expansion coefficient from aluminium [1/K]*)
  // print unit
  cPrintUnitTempCoefficient : LREAL := 17.3E-6; (*thermal expansion coefficient from print unit base plate [1/K]*)
  fC_PhPixelDistFactorAtRefTemp: LREAL := 0.1693/4;(*RICOH GEN5 PH pixel distance [mm] y direction of one pixel at reference temperature (instead of native resolution 600dpi)*)
  fC_PhPixelDistRefTemp     : LREAL := 23;      (*RICOH GEN5 PH reference temperature matching the fC_PhPixelDistFactorAtRefTemp*)

  // test telegram definitions
  sQvTest_Header            : STRING := 'QT_'; // qualivision test telegram header
  sQvTest_CI                : STRING := 'CI_'; // input frame timing test
  sQvTest_Loop              : STRING := 'LP_'; // loop timing test
  
  // debug
  nC_MaxRxTimingEntries     : UDINT := 40;
END_VAR

VAR PERSISTENT
  fCameraResolution         : LREAL := cCameraResolution;  (*Camera pixel resolution [dpi]*)
  fCameraAdjustmentY        : LREAL := 0;            (*Camera adjustment in Y direction [mm]*)
  fCameraCalTemp            : LREAL := 25;           (*calibration temperature for the given line camera resolution*)    
  fCameraStartMargin        : LREAL := 0.0085;       (*cM: Camera start margin [m]*)
END_VAR

// - live configuration update & checks
// -- trigger, cam position and trigger settings (Worker position setup)
_fTriggerDistance    := _fDetectToCameraOffset - fCameraStartMargin;
IF IfSpeed <> 0 THEN
  _fTriggerPulseLength := (fSubstrateLength + 2*fCameraStartMargin) / IfSpeed * 1000;  (*[ms] Margin at start and end of the sheet*)
END_IF

// --
IF fCameraResolution > 0 THEN
  fCameraWidthTC := DINT_TO_LREAL(_nCameraWidth) / fCameraResolution * 0.0254;
ELSE
  fCameraWidthTC := FC_CONV_SUBPX_TO_M( _nCameraWidth, LREAL_TO_UDINT(cCameraResolution), 1);
END_IF;

(*Camera temperature compensation (y-pos, center and resolution)*)
fCameraTemp             := INT_TO_LREAL(InTempActValueScanner) * 0.1;
fCameraDeltaTempFactor  := 1 + (cCameraTempCoefficient * (fCameraTemp - fCameraCalTemp));
fCameraRealResolution   := fCameraResolution / fCameraDeltaTempFactor; 
fCameraMechOffsetTAct   := _fCameraMechOffsetTC * fCameraDeltaTempFactor;
fCameraCenterOffsetTAct := (((fCameraWidthTC / 2 * 1000) + _fCameraMechOffsetTC) * fCameraDeltaTempFactor) - ((fCameraWidthTC / 2 * 1000) + _fCameraMechOffsetTC);

fPrintUnitTemp             := INT_TO_LREAL(InTempActValuePrintUnit) * 0.1;
fPrintUnitDeltaTempFactor  := 1 + (cPrintUnitTempCoefficient * (fPrintUnitTemp - _fPrintUnitCalTemp));
fPrintUnitMechOffsetTAct   := _fPrintUnitMechOffsetTC * fPrintUnitDeltaTempFactor;
fPrintUnitWidthTAct        := _fPrintUnitWidthTC * fPrintUnitDeltaTempFactor;

fPrintUnitWidthDiff        := fPrintUnitWidthTAct - _fPrintUnitWidthTC;
fPrintUnitCenterOffsetTAct := (((_fPrintUnitWidthTC / 2 * 1000) + _fPrintUnitMechOffsetTC) * fPrintUnitDeltaTempFactor) - ((_fPrintUnitWidthTC / 2 * 1000) + _fPrintUnitMechOffsetTC);

SimUpdate();

// Messages
(*fbMsg_NotEnoughTeachPoints( bI_Status:=SEL(_bActivated, FALSE, bNotEnoughTeachPoints), 
                             iI_MsgNumber:=eC_STAG_CAM_NOTENGOUGH_TEACH_POINTS, 
                             iI_MsgLocation:=ePr_BLK_CAMERA,
                             pI_MsgConfig:=_pMsgConfig);
*)

METHOD PRIVATE binarySearch : DINT
VAR_INPUT
  nLow : DINT;     // range lower
  nHigh : DINT;    // range upper
  nKey  : DINT;    // key to search
END_VAR
VAR
  mid : DINT;
END_VAR
IF nHigh < nLow THEN
  binarySearch := -1;
  RETURN;
END_IF

// split array in half
mid := (nLow + nHigh) / 2; (*low + (high - low)/2;*)

// did we find it?
IF nKey = TO_DINT(sTeachPoints[mid].id) THEN
  binarySearch := mid;
  RETURN;
END_IF

// no, search upper half (recursive)
IF nKey > TO_DINT(sTeachPoints[mid].id) THEN
  binarySearch := THIS^.binarySearch((mid + 1), nHigh, nKey);
  RETURN;
END_IF

// no, search lower half (recursive)
binarySearch:= THIS^.binarySearch(nLow, (mid - 1), nKey);
END_METHOD

{attribute 'monitoring' := 'call'}
(*Simulation is enabled set/get*)
PROPERTY bSimEnable : BOOL
GET
bSimEnable:=_bSimulate;
END_GET
SET
_bSimulate:=bSimEnable;
END_SET
END_PROPERTY

(*
  Calculate teached/saved reference points in print system coordinates.
*)
METHOD PRIVATE calcTeachPoints
VAR
  nCounter  : UDINT;
  nCurrSect : DINT;
  x_ref_abs : LREAL;
  y_ref_abs : LREAL;
  sTP       : ST_TeachPoint;
  sTPSend   : ST_DeformationPointAccurate;
END_VAR
IF _bVerbose THEN LogLvl(Lvl:=E_LogSeverity.Debug, Msg:='calculateTeachPoints()'); END_IF

bInvalidTeachPointsReceived := FALSE;

(*-- sort list with camera/teach points for faster binary searching later*)
sortPoints();

(*-- convert & save teach point in table separate table for later use*)
FOR nCounter := 1 TO nNbMarksTeach DO
  //--- save id
  sTP.id := sCameraPoints[nCounter].id;
  sTP.valid := sCameraPoints[nCounter].valid;
  
  //--- translate to print system coordinate system 
  IF (sCameraPoints[nCounter].x_ref = 0) THEN
    (*Fully automatic mode: ref value from camera is zero, ref value for printer is set with x.*)
    sTP.y_ref_Print   :=   ((_fPrintUnitWidthTC/2 + _fCameraWidthNormal/2) * 1000)  (*[m] => [mm]*)
                         - (  DINT_TO_REAL(sCameraPoints[nCounter].x)
                            / (cCameraResolution * cCameraResolutionSubpixel) * 25.4)           (*[mm]*)
                         - ((_fCameraWidthNormal - LREAL_TO_REAL(_fImageWidth)) * 1000 / 2);     (*[m] => [mm]*)
    sTP.y_teach_Print := 0;
  ELSE
    (*Semi automatic mode: ref value for printer is calculated with ref value and lx from camera.*)
    sTP.y_ref_Print   :=   (DINT_TO_REAL(sCameraPoints[nCounter].x_ref  - sCameraPoints[nCounter].lx)
                                      / (fCameraRealResolution * cCameraResolutionSubpixel) * 25.4);  (*[mm]*)
    sTP.y_teach_Print :=   (DINT_TO_REAL(sCameraPoints[nCounter].x)
                                      / (fCameraRealResolution * cCameraResolutionSubpixel) * 25.4);  (*[mm]*)
  END_IF
  
  IF (sCameraPoints[nCounter].y_ref = 0) THEN
    (*Fully automatic mode: ref value from camera is zero, ref value for printer is set with y.*)
    sTP.x_ref_Print   :=   (FC_CONV_SUBPX_TO_M( sCameraPoints[nCounter].y
                                              , LREAL_TO_UDINT(cCameraResolution)
                                              , LREAL_TO_UDINT(cCameraResolutionSubpixel)) * 1000)  (*[m] => [mm]*)
                         + (fCameraStartMargin * 1000);  (*[m] => [mm]*)
    sTP.x_teach_Print := 0;
  ELSE
    (*Semi automatic mode: ref value for printer is calculated with ref value and ly from camera.*)
    sTP.x_ref_Print   :=   (FC_CONV_SUBPX_TO_M( (sCameraPoints[nCounter].y_ref - sCameraPoints[nCounter].ly)
                                              , LREAL_TO_UDINT(cCameraResolution)
                                              , LREAL_TO_UDINT(cCameraResolutionSubpixel)) * 1000);  (*[m] => [mm]*)
    sTP.x_teach_Print :=   (FC_CONV_SUBPX_TO_M( sCameraPoints[nCounter].y
                                              , LREAL_TO_UDINT(cCameraResolution)
                                              , LREAL_TO_UDINT(cCameraResolutionSubpixel)) * 1000);  (*[m] => [mm]*)
  END_IF;
  
  //--- save teach point locally to seperate teach point array (the other one will be used for cam points while receiving) 
  sTeachPoints[nCounter] := sTP;
  
  //--- count points per sector (for error handling)
  IF (sTP.x_teach_Print = 0) THEN    (*Fully Automatic*)
    x_ref_abs := sTP.x_ref_Print;
  ELSE                                           (*Semi-automatic*)        
    x_ref_abs := sTP.x_ref_Print + sTP.x_teach_Print; 
  END_IF
  IF (sTP.y_teach_Print = 0) THEN    (*Fully Automatic*)
    y_ref_abs := sTP.y_ref_Print;
  ELSE                                           (*Semi-automatic*)        
    y_ref_abs := sTP.y_ref_Print + sTP.y_teach_Print;
  END_IF
  
  IF _fFrameLength <> 0 THEN
    nCurrSect := FC_LREAL_TO_DINT(x_ref_abs / _fFrameLength) + 1;
    nNumPointsPerSectorT[nCurrSect] := nNumPointsPerSectorT[nCurrSect] + 1;
  END_IF
  
  //--- send teach point to sink (python script)
  IF _iCameraSink <> 0 THEN
    sTPSend.x_ref := x_ref_abs;
    sTPSend.y_ref := y_ref_abs;
    sTPSend.dx    := 0;
    sTPSend.dy    := 0;
    sTPSend.col := nNumPointsPerSectorT[nCurrSect];  // point number in frame
    sTPSend.row := nCurrSect;                        // frame number
    _iCameraSink.AddTeachPoint(sTeachPoint:=sTPSend);
  END_IF
  
  //--- check if every teach point is valid
  IF NOT sTP.valid THEN
    bInvalidTeachPointsReceived := TRUE;
	END_IF
  
END_FOR

// verify the teach
verifyTeachPoints();
END_METHOD

METHOD CamTrigger
VAR_INPUT
  bOk             : BOOL;     // trigger is ok
	nPos            : DINT;     // camera triggered position
  nPosDeviation   : DINT;     // camera started deviation
  nX0             : DINT;     // detected position sheet/repetition
END_VAR
SUPER^.CamTrigger(bOk:=bOk, nPos:=nPos, nPosDeviation:=nPosDeviation, nX0:=nX0);

_tTimeTrigger := F_GetCurDcTaskTime64();    // save trigger time stamp (a little later than the real)
IF _bVerbose THEN LogLvl(Lvl:=E_LogSeverity.Debug, Msg:=F_Concat2('CamTrigger at: ', TO_STRING(_tTimeTrigger))); END_IF
nNbMarksScanned := 0;
END_METHOD

METHOD CamTriggerDone
SUPER^.CamTriggerDone();
IF _bVerbose THEN LogLvl(Lvl:=E_LogSeverity.Debug, Msg:=F_Concat2('CamTriggerDone at: ', TO_STRING(_tTimeTrigger))); END_IF
SimExit();
END_METHOD

(*
  Simulate camera points.
*)
METHOD PRIVATE CreateSimCamPoints : BOOL
VAR
  fbTonTimer     : TON;
  nCounter       : UDINT;
  nCamGridHeight : UDINT;    // cam points pitch in y in [px]
  nCamGridDepth  : UDINT;
  nIndex         : UDINT;
  nOffsetY       : UDINT;
  nCtr           : UDINT;
END_VAR
nCamGridDepth := _nSimCamFrameDepth;
nNbMarksTeach := _nSimCamMarksPerFrame * TO_UDINT((SEL(fSubstrateLength<>0, 5*nCamGridDepth, DINT_TO_UDINT(F_MeterToSubPixel(fPosMeter:=fSubstrateLength, fResoSubPx:=_nPrintUnitResolution)))) / nCamGridDepth);
nCamGridHeight := SEL(fSubstrateWidth<>0, 200, DINT_TO_UDINT(F_MeterToSubPixel(fPosMeter:=fSubstrateWidth, fResoSubPx:=_nPrintUnitResolution))/_nSimCamMarksPerFrame);
_bTeachOk := TRUE;

(*Test points*)
nCtr := 0;
nNbMarks := nNbMarksTeach;
nOffsetY := (_nPrintUnitWidthNormal-TO_UDINT(F_MeterToSubPixel(fPosMeter:=_fImageWidth, fResoSubPx:=_nPrintUnitResolution)))/2;

FOR nCounter := 0 TO nNbMarksTeach/_nSimCamMarksPerFrame - 1 DO    // col
  FOR nIndex := 0 TO _nSimCamMarksPerFrame-1 DO  // row
    // create point
    stCamPoint := getSimCamPoint(
      fOffsetMin:=-5.0,
      fOffsetMax:=5.0,
      fXMin:=nCounter*nCamGridDepth,
      fXMax:=(nCounter+1)*nCamGridDepth,
      fYMin:=nIndex*nCamGridHeight+nOffsetY,
      fYMax:=(nIndex+1)*nCamGridHeight+nOffsetY
    );
    // save simulation cam point
    nCtr := nCtr + 1;
    stCamPoint.index := TO_DINT(nCtr);
    stCamPoint.col   := TO_DINT(nCounter);
    stCamPoint.row   := TO_DINT(nIndex);
    _sSimCamPoints[nCtr] := stCamPoint;
  END_FOR
END_FOR
END_METHOD

{attribute 'monitoring':='call'}
PROPERTY eCameraMode : E_CameraMode
GET
// return active mode (after teach or live
eCameraMode := _eCameraMode;  // mode set by PUC

IF    _eCameraMode = E_CameraMode.Auto THEN
  eCameraMode := _ePossibleMode;
ELSIF _ePossibleMode < _eCameraMode THEN
  // reduced level
  eCameraMode := _ePossibleMode;
END_IF
END_GET
END_PROPERTY

PROPERTY eDeviceType : E_CameraDevice
GET
eDeviceType := E_CameraDevice.Scanner;
END_GET
END_PROPERTY

(*
  :return: CamReady 
*)
METHOD GetCamStatus : BOOL
VAR_OUTPUT
  bConnectionOK  : BOOL;    // Camera connected
  bTeachOk       : BOOL;    // Teach successful
  nTeachedPoints : UDINT;   // Teached points for this job
  nScannedPoints : UDINT;   // Scanned points on current sheet  
  bCamStarted    : BOOL;    // Camera trigger is active, cam started
  bCamDone       : BOOL;    // Camera finished on CT
  bErrors        : ARRAY[1..GVL_Camera.nC_NbCamErrors] OF BOOL;  // generic error flag list
END_VAR
bConnectionOK  := NOT bConnectionErr OR bSimulate;
bTeachOk       := _bTeachOk OR bSimulate;
nTeachedPoints := nNbMarksTeach;
nScannedPoints := nNbMarksScanned;
bCamStarted    := _bCamTriggerStarted;
// camera finished
IF nNbVersion = cProtoVersion_110 THEN
  // Done: Trigger released and last sector was received
  bCamDone       := _bCamTriggerDone AND ((nSector >= nNbSectorTeach) OR (nSector = SINT_TO_DINT(-1)));
ELSE
  // Done: Trigger released and same all teached points are scanned // NOTE: this will not work if not all marks are detected by camera
  bCamDone       := _bCamTriggerDone AND (nScannedPoints>=nTeachedPoints);
END_IF
GetCamStatus := bConnectionOK AND bTeachOk;   // camera ready
END_METHOD

(*
  get array index to point ID in stored point table
  :returns: TRUE if found, FALSE else
*)
METHOD getPointIndex : BOOL
VAR_INPUT
  nId : UDINT;
END_VAR
VAR_OUTPUT
  nIndex : UDINT;
END_VAR
VAR
  nResultIdx : DINT;
END_VAR
// search corresponding point in table (search for same mark ID)

nResultIdx := binarySearch(1, TO_DINT(nNbMarksTeach), TO_DINT(nId));
IF nResultIdx = -1 THEN
  LogWarning(F_Concat3('Point with Id: ', TO_STRING(nId) , ' not found in saved teach points'));
  nIndex := 1;
  RETURN;
END_IF

nIndex := TO_UDINT(nResultIdx);
getPointIndex := TRUE;
END_METHOD

METHOD INTERNAL getSimCamPoint : ST_DeformationPointAccurate
VAR_INPUT
  fXMin : LREAL := 0.0;
	fXMax : LREAL := 0.0;
	fYMin : LREAL := 0.0;
	fYMax : LREAL := 0.0;
	
	fOffsetMin : LREAL := 0.0;
	fOffsetMax : LREAL := 0.0;
END_VAR
VAR_OUTPUT
  sO_CamPoint : ST_DeformationPointAccurate;
END_VAR
VAR_INST
  fbRand : DRAND;
END_VAR
fbRand();
sO_CamPoint.x_ref := (fXMin + (fXMax - fXMin));
fbRand();
sO_CamPoint.y_ref := (fYMin + (fYMax - fYMin));

fbRand();
sO_CamPoint.dx := (fOffsetMin + (fOffsetMax - fOffsetMin) * fbRand.Num);
fbRand();
sO_CamPoint.dy := (fOffsetMin + (fOffsetMax - fOffsetMin) * fbRand.Num);

sO_CamPoint.valid := _bSimCamPointValid;
getSimCamPoint := sO_CamPoint;
END_METHOD

METHOD InitLineCamera
VAR_INPUT
  nPrintUnitResolution         : UDINT;    (*printhead pixel resolution [dpi]*)
  nPrintUnitSubPx              : UDINT;    (*print unit subPixel resolution [SubPx]*)
  nPrintUnitWidth              : UDINT;    (*print unit width in [px]*)
  iCameraTrigger               : I_CameraTrigger;
END_VAR
_fCameraWidthNormal     := FC_CONV_SUBPX_TO_M( _nCameraWidth
                                             , LREAL_TO_UDINT(cCameraResolution)
                                             , 1);
_nPrintUnitWidthNormal  := nPrintUnitWidth;
_fPrintUnitCalTemp      := fC_PhPixelDistRefTemp;   // reference temperate for real pixel spacing of ph
_fPrintUnitWidthTC      := (nPrintUnitWidth * fC_PhPixelDistFactorAtRefTemp) / 1000;  // caluclate print unit with at calibration temperature [m]

SUPER^.Init( nPrintUnitResolution:=nPrintUnitResolution
           , nPrintUnitSubPx:=nPrintUnitSubPx
           , iCameraTrigger := iCameraTrigger
           , bUseCameraTrigger:=TRUE
           , bUseCameraTriggerFeedback:=TRUE);
END_METHOD

METHOD InitSimulation : BOOL
VAR_INPUT
  aCamSimScriptPath : T_MaxString;
END_VAR
_aCamSimScriptPath := aCamSimScriptPath;
END_METHOD

METHOD mJobStart : BOOL
// re-calculate teach points with previous received 'T' telegram 
//  handles case: teach telegram arrived before JobStart
IF sModus = 'T' THEN calcTeachPoints(); END_IF
END_METHOD

(*
  Tcpip client rx message callback. 
  Called by FB_TcpMsgNotifier, registered with 'registerTcpIpClient()' before.
*)
METHOD rx_callback
VAR_INPUT
  sMessage : CalmarCompTcpIp.ST_TcpMsg;    // rx message
END_VAR
VAR
  sAnalyzeLastMessage    : STRING(GVL_TcpIp.TCP_RXDATA_SIZE);          // telegram string for analysis
  sTmpCamPoint           : ST_CameraPoint;
  
  nCounter               : UDINT;
  bOk, bEnd              : BOOL;

END_VAR
// basic message handling
SUPER^.rx_callback(sMessage := sMessage);
// debug print
IF _bVerbose THEN LogLvl(Lvl:=E_LogSeverity.Debug,Msg:=F_Concat4('Rx Sz: ', TO_STRING(nLastMessageSz), ' Msg:', sLastMessage)); END_IF

// check parameter (avoids crash)
IF _fPrintUnitWidthTC = 0 THEN LogError('rx_callback: Invalid configuration, review persistences and config values!'); RETURN; END_IF

// copy for parsing
sAnalyzeLastMessage := sLastMessage;      

REPEAT
  (*--- check message type ---*)
  // -- Is it a test message?
  IF rx_TestMsg(pMessage:=ADR(sLastMessage)) THEN       (*Test message*)
    RETURN;   // test message, ignore rest of parsing
   
  // -- Is it a error message ?
  ELSIF rx_ErrorMsg(pMessage:=ADR(sLastMessage)) THEN   (*Error message*)
    RETURN;   // error message, ignore rest of parsing
  
  // -- Is it a position message ('T' Teach or 'A' Auswertung)
  ELSIF rx_ParseHeader( pAnalyzeLastMessage := ADR(sAnalyzeLastMessage)
                      , nNbVersion      => nNbVersion          (*version*)
                      , sModus          => sModus              (*modus*)
                      , nNbMarks        => nNbMarks            (*number of marks*)
                      , nSector         => nSector)            (*sector*)
    THEN
     // got a position message, do not exit and do rest of parsing below
     // >>> DO parsing below 
     ;
    
  // -- unknown message
  ELSE
    IF _bVerbose THEN LogLvl(Lvl:=E_LogSeverity.Debug, Msg:=F_Concat2('unknown rx message (ignore): ', sLastMessage)); END_IF
    RETURN;
  END_IF
  
  
  (*--- Handle position telegram ---*)
  IF (sModus  = 'T') THEN 
    (*-- 'T' Teach message *)
    nNbMarksTeach   := 0;
    nNbMarksScanned := 0;
    nNbSectorTeach  := nSector;  (*Total number or sectors are send with teach message.*)
    sTeach          := sAnalyzeLastMessage; // display on visu
    
    IF _bVerbose THEN LogLvl(Lvl:=E_LogSeverity.Debug, Msg:='receive T telegram, erase cam/teach points list'); END_IF    
    MEMSET(destAddr:=ADR(sTeachPoints),  fillByte:=0, n:=SIZEOF(sTeachPoints));   // eraase teach points list
    MEMSET(destAddr:=ADR(sCameraPoints), fillByte:=0, n:=SIZEOF(sCameraPoints));  // erase cam points list
    MEMSET(destAddr:=ADR(nNumPointsPerSectorA), fillByte:=0, n:=SIZEOF(nNumPointsPerSectorA));
    MEMSET(destAddr:=ADR(nNumPointsPerSectorT), fillByte:=0, n:=SIZEOF(nNumPointsPerSectorT));
  ELSE
    (*-- 'A' Auswertung message *)
    sMemLastMessage := sAnalyzeLastMessage; // display on visu
    
    IF nSector = TO_DINT(cIdxFirstSector) THEN  // erase campoint with first received sector
      MEMSET(destAddr:=ADR(sCameraPoints), fillByte:=0, n:=SIZEOF(sCameraPoints));  // erase cam points list
      IF _bVerbose THEN LogLvl(Lvl:=E_LogSeverity.Debug, Msg:=F_Concat2('received first A sector, erase cam points list.','')); END_IF
      
      _nTimeFrameIdx_CamMsg := 1;
    END_IF
  
    // debug timing rx A
    IF _nTimeFrameIdx_CamMsg <= nC_MaxRxTimingEntries THEN  // save message timestamp for debugging
      _tTimeFrames_CamMsg[_nTimeFrameIdx_CamMsg] := F_GetCurDcTaskTime64();     // save cam frame rx timestamp
      _tTimeFramesMs_CamMsg[_nTimeFrameIdx_CamMsg] := TO_LREAL((_tTimeFrames_CamMsg[_nTimeFrameIdx_CamMsg]-_tTimeTrigger)/EC_DCTIME_TICKSPERMSEC64);  // delta to trigger in ms
      IF _bVerbose THEN 
        // dbg log rx frames
        LogLvl(Lvl:=E_LogSeverity.Debug, Msg:=F_Concat4(
            F_Concat2('A-Frame: ', TO_STRING(_nTimeFrameIdx_CamMsg)),
            F_Concat2(' : ', TO_STRING(_nTimeFrameIdx_CamMsg)),
            F_Concat2(' after trig: ', TO_STRING(_tTimeFramesMs_CamMsg[_nTimeFrameIdx_CamMsg])),
            F_Concat2(' at: ', TO_STRING(_tTimeFrames_CamMsg[_nTimeFrameIdx_CamMsg]))
        ));
			END_IF
      _nTimeFrameIdx_CamMsg := _nTimeFrameIdx_CamMsg + 1;
    END_IF
    
  END_IF;
  
  
  (*Search for rx, ry, lx, ly, v, x and y*)
  FOR nCounter := 1 TO nNbMarks DO
    // get next point
    IF NOT rx_ParsePoint(pAnalyzeLastMessage:=ADR(sAnalyzeLastMessage), sCamResult=>sTmpCamPoint, bLast=>bEnd) THEN 
      // invalid point received
      LogWarning(F_Concat2(
        F_Concat3('invalid ', SEL(sModus='T', 'camera', 'teach'), ' point received, '),
        F_CamPoint_ToString(sPoint:=sTmpCamPoint)
      ));
    END_IF
    IF bEnd AND nCounter < nNbMarks THEN LogWarning(F_Concat4('Less marks received than indicated in header: ', TO_STRING(nCounter), '<', TO_STRING(nNbMarks))); END_IF
    
    IF (sModus  = 'T') THEN
      (*-- 'T' Teach message *)
      // save (convert with job start)
      saveTeachPoint(sCamPoint := sTmpCamPoint);
    ELSE
      (*-- 'A' Auswertung message *)
      // save & convert cam point
      stCamPoint := saveAuswertungPoint(sCamPoint:=sTmpCamPoint, bOK=>bOk);     
      // stream point (if valid)
      IF bOk THEN  //AND sTmpCamPoint.valid THEN
        IF _iCameraSink <> 0 THEN
          _iCameraSink.AddCamPoint(stCamPoint);
          IF _bVerbose THEN 
            LogLvl(Lvl:=E_LogSeverity.Debug, Msg:= F_Concat2('AddCamPoint: ', F_DeformationPointAcc_ToString(sPointAcc:=stCamPoint)));
          END_IF
        END_IF
      END_IF
    END_IF
  END_FOR
UNTIL FIND2(ADR(sAnalyzeLastMessage), ADR(cStartString)) = 0   (*Search for another start string*)
END_REPEAT

IF (sModus  = 'T') THEN calcTeachPoints(); END_IF  // calculate teach points if it was a teach

bMsgReceived := FALSE;
END_METHOD

METHOD PRIVATE rx_DeleteMsgPart
VAR_INPUT
  pAnalyzeLastMessage    : POINTER TO STRING(GVL_TcpIp.TCP_RXDATA_SIZE);  // telegram string for analysis
  nLen                   : UDINT;
  nPos                   : UDINT;
END_VAR
VAR
  sMessageDelete         : STRING(GVL_TcpIp.TCP_RXDATA_SIZE);             // telegram string for analysis
END_VAR
DELETE2( pSrcString := pAnalyzeLastMessage
       , pDstString := ADR(sMessageDelete)
       , nDstSize   := SIZEOF(sMessageDelete)
       , nLen       := nLen
       , nPos       := nPos);

pAnalyzeLastMessage^ := sMessageDelete;
END_METHOD

(*
  Parse for error message
  :return: TRUE if it was an error test telegram, FALSE if other.
*)
METHOD PRIVATE rx_ErrorMsg : BOOL
VAR_INPUT
  pMessage    : POINTER TO STRING(GVL_TcpIp.TCP_RXDATA_SIZE);   // tcp message string pointer 
END_VAR
VAR
  nFIdx : UDINT;    // string find index
  nFrmIdx : UDINT;
  tDiff : LREAL;
  sErrMsg : T_MaxString;
END_VAR
// parse message type
nFIdx := FIND2(pMessage, ADR(cErrorString));
IF nFIdx > 0 THEN  
  IF _bVerbose THEN LogLvl(Lvl:=E_LogSeverity.Debug, Msg:=F_Concat2('error: msg received: ', pMessage^)); END_IF

  // error telegram received
  DELETE2( pSrcString := pMessage
         , pDstString := ADR(sErrMsg)
         , nDstSize   := SIZEOF(sErrMsg)
         , nLen       := (nFIdx + INT_TO_UDINT(LEN(cErrorString)) - 1)
         , nPos       := 1);

  // strip other control characters
  FindAndDelete(pSrcString:=ADR(sErrMsg), pDstString:=ADR(sErrMsg), nDstSize:=SIZEOF(sErrMsg), pDeleteString:=ADR(cEndingString));
  
  // error message implement handling
  
  rx_ErrorMsg := TRUE;
ELSE
  ; // other telegram
END_IF
END_METHOD

(*
  Parse for position telegram header.
  :return: TRUE if valid position telegram, FALSE else
*)
METHOD PRIVATE rx_ParseHeader : BOOL
VAR_INPUT
  pAnalyzeLastMessage    : POINTER TO STRING(GVL_TcpIp.TCP_RXDATA_SIZE);  // telegram string for analysis
END_VAR
VAR_OUTPUT
  nNbVersion             : INT;                   (*(V) Version: protocol version, e.g. 100/110/...*)
  sModus                 : T_MaxString;           (*(M) Modus: 'T'/'A'*)
  nNbMarks               : UDINT;                 (*(A) Merkmale: number of Marks in Teach/Auswertung*)
  nSector                : DINT;                  (*(S) Sectors: Number of Sectors in 'T' / Sector index in 'A'*)
  //sMemLastMessage        : STRING(GVL_TcpIp.TCP_RXDATA_SIZE);  (*rx telegram string without header*)
END_VAR
VAR
  nFindIndex             : UDINT;
END_VAR
(*Search for start string*)
nFindIndex := FIND2(pAnalyzeLastMessage, ADR(cStartString));
IF nFindIndex = 0 THEN RETURN; END_IF

(*Search string found => remove string to evaluate rest of message*)
rx_DeleteMsgPart(pAnalyzeLastMessage := pAnalyzeLastMessage, nLen := (nFindIndex + INT_TO_UDINT(LEN(cStartString)) - 1) , nPos := 1);

(*Search for version number*)
nFindIndex := FIND2(pAnalyzeLastMessage, ADR(','));
IF nFindIndex > 0 THEN
  nNbVersion := STRING_TO_INT(LEFT(pAnalyzeLastMessage^, (UDINT_TO_INT(nFindIndex) - 1)));

  rx_DeleteMsgPart(pAnalyzeLastMessage := pAnalyzeLastMessage, nLen := nFindIndex , nPos := 1);
END_IF;

(*Search for modus (M)*)
nFindIndex := FIND2(pAnalyzeLastMessage, ADR(','));
IF nFindIndex > 0 THEN
  sModus := LEFT(pAnalyzeLastMessage^, (UDINT_TO_INT(nFindIndex) - 1));

  rx_DeleteMsgPart(pAnalyzeLastMessage := pAnalyzeLastMessage, nLen := nFindIndex , nPos := 1);
END_IF;

(*Search for number marks (A)*)
nFindIndex := FIND2(pAnalyzeLastMessage, ADR(','));
IF nFindIndex > 0 THEN
  nNbMarks := STRING_TO_UDINT(LEFT(pAnalyzeLastMessage^, (UDINT_TO_INT(nFindIndex) - 1)));
  IF nNbMarks > GVL_Camera.cMaxNbMarks THEN
    LogLvl(Lvl:=E_LogSeverity.Warning, Msg:=F_Concat4('Limit marks (', TO_STRING(nNbMarks),') to max=', TO_STRING(GVL_Camera.cMaxNbMarks)));
    nNbMarks := GVL_Camera.cMaxNbMarks;
  END_IF

  rx_DeleteMsgPart(pAnalyzeLastMessage := pAnalyzeLastMessage, nLen := nFindIndex , nPos := 1);
END_IF;

(*Search for sector of transmission (S)*)
nFindIndex := FIND2(pAnalyzeLastMessage, ADR(','));
IF nFindIndex > 0 THEN
  (*Last sector is indicated with '-1'*)
  nSector := STRING_TO_DINT(LEFT(pAnalyzeLastMessage^, (UDINT_TO_INT(nFindIndex) - 1)));

